C03580=1008.625,303.461,-161.555,-20.052,46.107,35.019
C03581=1008.519,303.701,-161.743,-19.485,46.587,36.235
C03582=1008.413,303.937,-161.933,-18.890,47.066,37.479
C03583=1008.305,304.173,-162.124,-18.265,47.545,38.750
C03584=1008.220,304.356,-162.274,-17.761,47.914,39.754
C03585=1008.136,304.538,-162.423,-17.237,48.283,40.777
C03586=1008.050,304.719,-162.574,-16.695,48.650,41.816
C03587=1007.964,304.899,-162.726,-16.132,49.015,42.875
C03588=1007.851,305.131,-162.923,-15.372,49.485,44.275
C03589=1007.738,305.362,-163.122,-14.578,49.950,45.708
C03590=1007.623,305.592,-163.322,-13.751,50.408,47.169
C03591=1007.508,305.821,-163.524,-12.888,50.859,48.662
C03592=1007.418,305.995,-163.679,-12.202,51.199,49.829
C03593=1007.328,306.169,-163.835,-11.496,51.534,51.012
C03594=1007.237,306.341,-163.992,-10.767,51.863,52.216
C03595=1007.147,306.513,-164.150,-10.017,52.187,53.438
C03596=1007.025,306.737,-164.358,-9.002,52.599,55.068
C03597=1006.905,306.961,-164.566,-7.948,53.000,56.733
C03598=1006.782,307.182,-164.777,-6.854,53.388,58.434
C03599=1006.659,307.402,-164.988,-5.724,53.761,60.165
C03600=1006.565,307.568,-165.150,-4.837,54.035,61.506
C03601=1006.470,307.733,-165.312,-3.930,54.299,62.863
C03602=1006.375,307.898,-165.475,-2.999,54.554,64.242
C03603=1006.278,308.061,-165.638,-2.047,54.798,65.640
C03604=1006.150,308.276,-165.856,-0.758,55.103,67.512
C03605=1006.021,308.489,-166.075,0.564,55.388,69.411
C03606=1005.891,308.702,-166.295,1.921,55.651,71.337
C03607=1005.760,308.912,-166.516,3.305,55.891,73.285
C03608=1005.653,309.083,-166.696,4.453,56.070,74.887
C03609=1005.546,309.251,-166.878,5.620,56.233,76.503
C03610=1005.908,309.402,-167.279,6.450,56.338,77.647
C03611=1006.056,309.174,-167.035,4.862,56.129,75.455
C03612=1006.201,308.944,-166.790,3.305,55.891,73.285
C03613=1006.331,308.733,-166.569,1.921,55.651,71.337
C03614=1006.462,308.522,-166.350,0.564,55.388,69.411
C03615=1006.591,308.308,-166.131,-0.758,55.103,67.512
C03616=1006.719,308.092,-165.913,-2.047,54.798,65.640
C03617=1006.815,307.929,-165.750,-2.999,54.554,64.242
C03618=1006.910,307.765,-165.587,-3.930,54.299,62.863
C03619=1007.005,307.600,-165.425,-4.837,54.035,61.506
C03620=1007.099,307.434,-165.263,-5.724,53.761,60.165
C03621=1007.223,307.214,-165.051,-6.854,53.388,58.434
C03622=1007.345,306.992,-164.841,-7.948,53.000,56.733
C03623=1007.467,306.769,-164.632,-9.002,52.599,55.068
C03624=1007.587,306.545,-164.424,-10.017,52.187,53.438
C03625=1007.677,306.373,-164.267,-10.767,51.863,52.216
C03626=1007.768,306.200,-164.110,-11.496,51.534,51.012
C03627=1007.858,306.027,-163.954,-12.202,51.199,49.829
C03628=1007.948,305.853,-163.798,-12.888,50.859,48.662
C03629=1008.064,305.623,-163.596,-13.751,50.408,47.169
C03630=1008.178,305.394,-163.396,-14.578,49.950,45.708
C03631=1008.291,305.163,-163.197,-15.372,49.485,44.275
C03632=1008.404,304.930,-163.000,-16.132,49.015,42.875
C03633=1008.490,304.750,-162.849,-16.695,48.650,41.816
C03634=1008.576,304.569,-162.698,-17.237,48.283,40.777
C03635=1008.661,304.388,-162.548,-17.761,47.914,39.754
C03636=1008.745,304.206,-162.398,-18.265,47.545,38.750
C03637=1008.853,303.969,-162.207,-18.890,47.066,37.479
C03638=1008.959,303.732,-162.018,-19.485,46.587,36.235
C03639=1009.065,303.494,-161.829,-20.052,46.107,35.019
C03640=1009.170,303.254,-161.642,-20.592,45.628,33.828
C03641=1009.251,303.066,-161.497,-20.996,45.254,32.916
C03642=1009.330,302.878,-161.352,-21.384,44.880,32.017
C03643=1009.410,302.689,-161.209,-21.757,44.508,31.133
C03644=1009.490,302.499,-161.066,-22.115,44.137,30.264
C03645=1009.590,302.256,-160.886,-22.552,43.665,29.173
C03646=1009.689,302.013,-160.706,-22.967,43.196,28.105
C03647=1009.787,301.768,-160.527,-23.359,42.732,27.060
C03648=1009.884,301.522,-160.351,-23.731,42.271,26.037
C03649=1009.959,301.327,-160.212,-24.010,41.911,25.245
C03650=1010.035,301.132,-160.075,-24.278,41.553,24.463
C03651=1010.110,300.936,-159.937,-24.533,41.199,23.695
C03652=1010.183,300.739,-159.802,-24.778,40.847,22.938
C03653=1010.276,300.491,-159.630,-25.071,40.409,21.999
C03654=1010.367,300.241,-159.461,-25.349,39.974,21.077
C03655=1010.458,299.990,-159.293,-25.610,39.546,20.172
///RCONF 0,0,0,0,1,0,0,0,0,0,0,0,0,0,0,0,0,0,0,0,0,0,0,0
C03656=1010.548,299.739,-159.127,-25.857,39.121,19.283
C03657=1010.618,299.539,-158.994,-26.044,38.788,18.586
C03658=1010.688,299.336,-158.863,-26.221,38.458,17.898
C03659=1010.757,299.135,-158.733,-26.391,38.132,17.220
C03660=1010.826,298.932,-158.604,-26.551,37.810,16.553
C03661=1010.911,298.678,-158.442,-26.741,37.414,15.733
C03662=1010.996,298.423,-158.283,-26.918,37.024,14.926
C03663=1011.079,298.168,-158.125,-27.085,36.641,14.134
C03664=1011.161,297.911,-157.968,-27.241,36.263,13.354
C03665=1011.228,297.705,-157.842,-27.359,35.965,12.738
C03666=1011.293,297.498,-157.718,-27.470,35.670,12.129
C03667=1011.357,297.290,-157.593,-27.576,35.380,11.529
C03668=1011.421,297.082,-157.470,-27.675,35.094,10.935
C03669=1011.499,296.824,-157.319,-27.790,34.746,10.213
C03670=1011.577,296.565,-157.169,-27.897,34.404,9.500
C03671=1011.653,296.305,-157.020,-27.996,34.069,8.801
C03672=1011.729,296.045,-156.872,-28.087,33.739,8.111
C03673=1011.789,295.834,-156.753,-28.156,33.478,7.560
C03674=1011.850,295.621,-156.636,-28.220,33.220,7.016
C03675=1011.910,295.408,-156.517,-28.280,32.966,6.479
C03676=1011.969,295.196,-156.400,-28.335,32.716,5.947
C03677=1012.041,294.934,-156.258,-28.398,32.417,5.306
C03678=1012.112,294.670,-156.117,-28.455,32.122,4.672
C03679=1012.182,294.408,-155.978,-28.506,31.835,4.050
C03680=1012.252,294.143,-155.838,-28.552,31.552,3.436
C03681=1012.308,293.928,-155.725,-28.586,31.327,2.940
C03682=1012.364,293.711,-155.613,-28.617,31.104,2.450
C03683=1012.419,293.493,-155.501,-28.645,30.886,1.967
C03684=1012.473,293.276,-155.391,-28.669,30.673,1.490
C03685=1012.539,293.010,-155.257,-28.695,30.417,0.916
C03686=1012.603,292.745,-155.124,-28.717,30.168,0.353
C03687=1012.668,292.479,-154.993,-28.736,29.926,-0.203
C03688=1012.731,292.212,-154.862,-28.751,29.686,-0.753
C03689=1012.783,291.992,-154.755,-28.760,29.494,-1.200
C03690=1012.834,291.771,-154.649,-28.768,29.306,-1.642
C03691=1012.885,291.550,-154.543,-28.773,29.120,-2.080
C03692=1012.935,291.329,-154.438,-28.777,28.937,-2.514
C03693=1012.996,291.061,-154.312,-28.778,28.722,-3.030
C03694=1013.054,290.793,-154.187,-28.777,28.512,-3.541
C03695=1013.113,290.524,-154.064,-28.773,28.305,-4.046
C03696=1013.171,290.255,-153.941,-28.767,28.103,-4.544
C03697=1013.219,290.031,-153.840,-28.760,27.939,-4.952
C03698=1013.265,289.806,-153.739,-28.752,27.779,-5.357
C03699=1013.312,289.582,-153.639,-28.742,27.622,-5.757
C03700=1013.358,289.357,-153.540,-28.730,27.467,-6.153
C03701=1013.413,289.087,-153.422,-28.715,27.285,-6.624
C03702=1013.467,288.817,-153.304,-28.698,27.109,-7.088
C03703=1013.520,288.545,-153.189,-28.679,26.937,-7.545
C03704=1013.573,288.274,-153.072,-28.659,26.767,-7.999
C03705=1013.617,288.047,-152.977,-28.641,26.630,-8.372
C03706=1013.660,287.819,-152.882,-28.622,26.495,-8.743
C03707=1013.701,287.592,-152.787,-28.602,26.363,-9.109
C03708=1013.744,287.364,-152.694,-28.581,26.233,-9.471
C03709=1013.794,287.092,-152.582,-28.555,26.082,-9.899
C03710=1013.842,286.820,-152.472,-28.527,25.935,-10.321
C03711=1013.890,286.547,-152.363,-28.499,25.792,-10.737
C03712=1013.938,286.275,-152.254,-28.470,25.652,-11.148
C03713=1013.978,286.044,-152.164,-28.444,25.537,-11.492
C03714=1014.017,285.814,-152.074,-28.418,25.425,-11.832
C03715=1014.056,285.584,-151.985,-28.391,25.314,-12.171
C03716=1014.094,285.354,-151.895,-28.364,25.204,-12.507
C03717=1014.139,285.080,-151.791,-28.330,25.079,-12.901
C03718=1014.183,284.807,-151.688,-28.296,24.956,-13.292
C03719=1014.227,284.533,-151.585,-28.261,24.835,-13.680
C03720=1014.270,284.258,-151.484,-28.226,24.716,-14.065
C03721=1014.306,284.026,-151.398,-28.195,24.619,-14.388
C03722=1014.341,283.794,-151.313,-28.164,24.524,-14.708
C03723=1014.377,283.561,-151.229,-28.132,24.429,-15.026
C03724=1014.411,283.328,-151.145,-28.100,24.338,-15.343
C03725=1014.451,283.053,-151.048,-28.062,24.232,-15.713
C03726=1014.490,282.778,-150.950,-28.023,24.128,-16.079
C03727=1014.530,282.504,-150.854,-27.984,24.027,-16.441
C03728=1014.568,282.228,-150.759,-27.945,23.929,-16.801
C03729=1014.600,281.993,-150.677,-27.911,23.848,-17.104
C03730=1014.633,281.758,-150.597,-27.877,23.768,-17.406
C03731=1014.663,281.524,-150.518,-27.842,23.690,-17.706
C03732=1014.695,281.288,-150.439,-27.807,23.613,-18.004
C03733=1014.731,281.013,-150.347,-27.766,23.526,-18.349
C03734=1014.766,280.737,-150.256,-27.725,23.440,-18.691
C03735=1014.800,280.461,-150.166,-27.684,23.357,-19.031
C03736=1014.835,280.185,-150.076,-27.642,23.276,-19.367
C03737=1014.863,279.948,-150.000,-27.606,23.208,-19.653
C03738=1014.892,279.711,-149.925,-27.570,23.143,-19.936
C03739=1014.920,279.474,-149.851,-27.534,23.078,-20.218
C03740=1014.948,279.238,-149.777,-27.498,23.014,-20.499
C03741=1014.980,278.961,-149.691,-27.456,22.942,-20.824
C03742=1015.011,278.685,-149.606,-27.413,22.872,-21.148
C03743=1015.042,278.408,-149.522,-27.370,22.804,-21.469
C03744=1015.072,278.131,-149.437,-27.327,22.737,-21.789
C03745=1015.097,277.892,-149.366,-27.290,22.681,-22.062
C03746=1015.122,277.654,-149.296,-27.252,22.626,-22.334
C03747=1015.148,277.415,-149.226,-27.215,22.573,-22.606
C03748=1015.172,277.176,-149.155,-27.177,22.521,-22.877
C03749=1015.199,276.899,-149.076,-27.134,22.462,-23.186
C03750=1015.226,276.622,-148.996,-27.090,22.404,-23.496
C03751=1015.253,276.345,-148.917,-27.046,22.349,-23.804
C03752=1015.279,276.068,-148.840,-27.003,22.295,-24.109
C03753=1015.301,275.828,-148.773,-26.965,22.250,-24.373
C03754=1015.323,275.588,-148.708,-26.927,22.204,-24.635
C03755=1015.344,275.347,-148.641,-26.889,22.162,-24.896
C03756=1015.366,275.107,-148.577,-26.851,22.119,-25.156
C03757=1015.390,274.829,-148.502,-26.807,22.073,-25.453
C03758=1015.412,274.552,-148.428,-26.763,22.027,-25.750
C03759=1015.435,274.275,-148.355,-26.720,21.983,-26.043
C03760=1015.458,273.996,-148.282,-26.676,21.940,-26.336
C03761=1015.477,273.755,-148.221,-26.638,21.904,-26.589
C03762=1015.496,273.513,-148.158,-26.600,21.869,-26.841
C03763=1015.513,273.271,-148.097,-26.562,21.835,-27.092
C03764=1015.532,273.030,-148.036,-26.525,21.803,-27.342
C03765=1015.551,272.752,-147.968,-26.481,21.766,-27.626
C03766=1015.571,272.474,-147.900,-26.438,21.731,-27.910
C03767=1015.591,272.196,-147.832,-26.395,21.697,-28.194
C03768=1015.609,271.918,-147.764,-26.351,21.664,-28.476
C03769=1015.625,271.674,-147.706,-26.314,21.637,-28.720
C03770=1015.640,271.432,-147.649,-26.276,21.610,-28.964
C03771=1015.656,271.188,-147.593,-26.238,21.585,-29.208
C03772=1015.670,270.945,-147.536,-26.201,21.560,-29.450
C03773=1015.685,270.668,-147.472,-26.158,21.533,-29.728
C03774=1015.703,270.389,-147.409,-26.115,21.507,-30.003
C03775=1015.718,270.111,-147.348,-26.072,21.483,-30.277
C03776=1015.732,269.832,-147.286,-26.030,21.459,-30.551
C03777=1015.746,269.588,-147.232,-25.992,21.438,-30.791
C03778=1015.757,269.344,-147.180,-25.955,21.420,-31.029
C03779=1015.769,269.100,-147.127,-25.918,21.402,-31.266
C03780=1015.781,268.856,-147.075,-25.881,21.386,-31.502
C03781=1015.794,268.577,-147.017,-25.839,21.367,-31.772
C03782=1015.806,268.299,-146.958,-25.797,21.350,-32.039
C03783=1015.818,268.021,-146.901,-25.755,21.334,-32.305
C03784=1015.829,267.742,-146.845,-25.714,21.319,-32.571
C03785=1015.839,267.497,-146.796,-25.677,21.306,-32.805
C03786=1015.848,267.251,-146.747,-25.641,21.295,-33.037
C03787=1015.857,267.006,-146.699,-25.604,21.284,-33.268
C03788=1015.866,266.760,-146.652,-25.568,21.275,-33.499
C03789=1015.875,266.482,-146.599,-25.527,21.264,-33.760
C03790=1015.883,266.203,-146.545,-25.487,21.254,-34.021
C03791=1015.891,265.925,-146.493,-25.446,21.246,-34.279
C03792=1015.899,265.646,-146.442,-25.406,21.239,-34.538
C03793=1015.905,265.399,-146.398,-25.370,21.233,-34.766
C03794=1015.912,265.154,-146.353,-25.335,21.229,-34.991
C03795=1015.918,264.908,-146.310,-25.300,21.225,-35.219
C03796=1015.924,264.661,-146.267,-25.265,21.221,-35.444
C03797=1015.929,264.383,-146.219,-25.226,21.219,-35.699
C03798=1015.934,264.103,-146.170,-25.186,21.217,-35.952
C03799=1015.939,263.824,-146.124,-25.147,21.216,-36.205
C03800=1015.943,263.545,-146.078,-25.108,21.215,-36.458
C03801=1015.947,263.298,-146.037,-25.074,21.216,-36.681
C03802=1015.950,263.051,-145.997,-25.040,21.217,-36.903
C03803=1015.953,262.804,-145.958,-25.006,21.220,-37.124
C03804=1015.955,262.558,-145.919,-24.973,21.223,-37.345
C03805=1015.957,262.278,-145.876,-24.935,21.227,-37.593
C03806=1015.959,261.999,-145.833,-24.897,21.233,-37.842
C03807=1015.961,261.719,-145.791,-24.860,21.238,-38.090
C03808=1015.961,261.440,-145.750,-24.823,21.245,-38.337
C03809=1015.962,261.192,-145.714,-24.790,21.251,-38.554
C03810=1015.962,260.945,-145.679,-24.758,21.259,-38.770
C03811=1015.962,260.698,-145.644,-24.725,21.267,-38.988
C03812=1015.961,260.451,-145.609,-24.693,21.275,-39.204
C03813=1015.960,260.171,-145.571,-24.658,21.287,-39.446
C03814=1015.958,259.891,-145.533,-24.622,21.298,-39.688
C03815=1015.957,259.612,-145.496,-24.587,21.310,-39.930
C03816=1015.954,259.332,-145.460,-24.551,21.322,-40.171
C03817=1015.938,258.096,-145.307,-24.430,21.375,-41.012
C03818=1015.934,257.852,-145.277,-24.430,21.375,-41.014
C03819=1015.931,257.609,-145.248,-24.429,21.375,-41.018
C03820=1015.928,257.366,-145.220,-24.429,21.376,-41.019
C03821=1015.925,257.122,-145.191,-24.429,21.376,-41.021
C03822=1015.922,256.879,-145.162,-24.428,21.375,-41.025
C03823=1015.919,256.635,-145.132,-24.428,21.376,-41.027
C03824=1015.915,256.392,-145.104,-24.428,21.377,-41.029
C03825=1015.912,256.144,-145.074,-24.427,21.376,-41.032
C03826=1015.908,255.895,-145.044,-24.427,21.376,-41.034
C03827=1015.905,255.648,-145.014,-24.426,21.376,-41.037
C03828=1015.901,255.399,-144.985,-24.426,21.377,-41.040
C03829=1015.899,255.151,-144.955,-24.426,21.377,-41.042
C03830=1015.895,254.903,-144.926,-24.425,21.377,-41.045
C03831=1015.892,254.654,-144.897,-24.425,21.377,-41.047
C03832=1015.889,254.406,-144.866,-24.425,21.377,-41.049
C03833=1015.885,254.158,-144.837,-24.424,21.378,-41.052
C03834=1015.882,253.909,-144.808,-24.424,21.378,-41.054
C03835=1015.879,253.661,-144.779,-24.424,21.378,-41.058
C03836=1015.876,253.414,-144.749,-24.423,21.378,-41.060
C03837=1015.872,253.165,-144.720,-24.423,21.378,-41.061
C03838=1015.870,252.917,-144.690,-24.423,21.378,-41.065
C03839=1015.866,252.668,-144.660,-24.422,21.379,-41.067
C03840=1015.863,252.420,-144.631,-24.422,21.379,-41.069
C03841=1015.860,252.172,-144.602,-24.421,21.378,-41.072
C03842=1015.857,251.923,-144.572,-24.421,21.379,-41.074
C03843=1015.854,251.675,-144.544,-24.421,21.380,-41.076
C03844=1015.850,251.427,-144.513,-24.421,21.380,-41.078
C03845=1015.847,251.184,-144.485,-24.420,21.380,-41.082
C03846=1015.844,250.940,-144.456,-24.420,21.380,-41.084
C03847=1015.841,250.697,-144.428,-24.420,21.380,-41.085
C03848=1015.838,250.454,-144.399,-24.419,21.380,-41.089
C03849=1015.835,250.211,-144.370,-24.419,21.380,-41.091
C03850=1015.831,249.968,-144.341,-24.419,21.381,-41.093
C03851=1015.829,249.724,-144.313,-24.418,21.381,-41.095
C03852=1015.826,249.480,-144.284,-24.418,21.381,-41.098
C03853=1015.823,249.232,-144.255,-24.418,21.381,-41.100
C03854=1015.819,248.984,-144.226,-24.417,21.381,-41.102
C03855=1015.816,248.735,-144.197,-24.417,21.381,-41.104
C03856=1015.813,248.488,-144.168,-24.417,21.381,-41.107
C03857=1015.810,248.240,-144.138,-24.416,21.381,-41.109
C03858=1015.807,247.992,-144.109,-24.416,21.382,-41.111
C03859=1015.804,247.743,-144.079,-24.416,21.382,-41.113
C03860=1015.800,247.495,-144.051,-24.415,21.382,-41.117
C03861=1015.798,247.247,-144.021,-24.415,21.382,-41.118
C03862=1015.795,246.999,-143.992,-24.415,21.382,-41.120
C03863=1015.792,246.750,-143.964,-24.414,21.383,-41.122
C03864=1015.789,246.501,-143.935,-24.414,21.382,-41.126
C03865=1015.786,246.253,-143.905,-24.414,21.382,-41.127
C03866=1015.783,246.005,-143.876,-24.413,21.383,-41.129
C03867=1015.780,245.757,-143.847,-24.413,21.384,-41.132
C03868=1015.777,245.509,-143.818,-24.413,21.384,-41.134
C03869=1015.773,245.260,-143.789,-24.412,21.384,-41.137
C03870=1015.771,245.012,-143.760,-24.412,21.384,-41.139
C03871=1015.767,244.764,-143.731,-24.412,21.384,-41.141
C03872=1015.765,244.515,-143.702,-24.412,21.384,-41.143
C03873=1015.762,244.279,-143.674,-24.411,21.384,-41.144
C03874=1015.759,244.041,-143.647,-24.411,21.384,-41.148
C03875=1015.756,243.804,-143.620,-24.411,21.384,-41.150
C03876=1015.754,243.567,-143.591,-24.410,21.384,-41.151
C03877=1015.751,243.330,-143.564,-24.410,21.385,-41.153
C03878=1015.748,243.093,-143.536,-24.410,21.385,-41.155
C03879=1015.745,242.857,-143.509,-24.410,21.385,-41.157
C03880=1015.742,242.619,-143.481,-24.409,21.385,-41.159
C03881=1015.739,242.371,-143.452,-24.409,21.386,-41.161
C03882=1015.736,242.123,-143.423,-24.408,21.385,-41.164
C03883=1015.734,241.874,-143.394,-24.408,21.385,-41.166
C03884=1015.731,241.626,-143.365,-24.408,21.386,-41.168
C03885=1015.728,241.378,-143.336,-24.408,21.386,-41.170
C03886=1015.725,241.129,-143.308,-24.407,21.386,-41.172
C03887=1015.723,240.881,-143.279,-24.407,21.386,-41.174
C03888=1015.719,240.633,-143.250,-24.407,21.386,-41.176
C03889=1015.717,240.385,-143.222,-24.406,21.386,-41.179
C03890=1015.714,240.136,-143.192,-24.406,21.386,-41.181
C03891=1015.711,239.888,-143.164,-24.406,21.386,-41.183
C03892=1015.709,239.639,-143.135,-24.406,21.387,-41.184
C03893=1015.706,239.379,-143.105,-24.405,21.387,-41.186
C03894=1015.702,239.118,-143.075,-24.405,21.387,-41.188
C03895=1015.699,238.858,-143.044,-24.405,21.387,-41.190
C03896=1015.696,238.597,-143.014,-24.405,21.388,-41.192
C03897=1015.694,238.348,-142.986,-24.404,21.387,-41.195
C03898=1015.691,238.100,-142.957,-24.404,21.387,-41.197
C03899=1015.688,237.852,-142.929,-24.403,21.388,-41.199
C03900=1015.686,237.604,-142.900,-24.403,21.388,-41.201
C03901=1015.683,237.360,-142.872,-24.403,21.388,-41.203
C03902=1015.680,237.117,-142.843,-24.403,21.388,-41.205
C03903=1015.677,236.874,-142.816,-24.402,21.388,-41.207
C03904=1015.675,236.631,-142.787,-24.402,21.389,-41.209
C03905=1015.672,236.388,-142.759,-24.402,21.389,-41.210
C03906=1015.670,236.145,-142.731,-24.402,21.389,-41.212
C03907=1015.667,235.902,-142.704,-24.401,21.389,-41.214
C03908=1015.664,235.659,-142.676,-24.401,21.390,-41.216
C03909=1015.662,235.410,-142.647,-24.401,21.389,-41.218
C03910=1015.658,235.162,-142.618,-24.401,21.389,-41.219
C03911=1015.656,234.914,-142.589,-24.400,21.389,-41.221
C03912=1015.653,234.665,-142.561,-24.400,21.390,-41.223
C03913=1015.651,234.418,-142.533,-24.400,21.390,-41.225
C03914=1015.648,234.169,-142.504,-24.400,21.390,-41.227
C03915=1015.645,233.921,-142.475,-24.399,21.390,-41.229
C03916=1015.643,233.672,-142.447,-24.399,21.390,-41.231
C03917=1015.640,233.423,-142.419,-24.399,21.391,-41.233
C03918=1015.638,233.176,-142.390,-24.399,21.391,-41.234
C03919=1015.635,232.927,-142.362,-24.398,21.391,-41.236
C03920=1015.632,232.679,-142.334,-24.398,21.390,-41.238
C03921=1015.630,232.430,-142.304,-24.398,21.391,-41.240
C03922=1015.627,232.182,-142.277,-24.397,21.391,-41.242
C03923=1015.625,231.933,-142.248,-24.397,21.391,-41.243
C03924=1015.622,231.685,-142.220,-24.397,21.391,-41.245
C03925=1015.619,231.437,-142.191,-24.397,21.392,-41.247
C03926=1015.617,231.189,-142.163,-24.396,21.392,-41.249
C03927=1015.614,230.940,-142.135,-24.396,21.392,-41.251
C03928=1015.612,230.691,-142.106,-24.396,21.391,-41.252
C03929=1015.609,230.449,-142.078,-24.396,21.392,-41.254
C03930=1015.607,230.206,-142.050,-24.395,21.392,-41.256
C03931=1015.605,229.963,-142.023,-24.395,21.392,-41.258
C03932=1015.602,229.720,-141.995,-24.395,21.392,-41.260
C03933=1015.600,229.476,-141.967,-24.395,21.392,-41.262
C03934=1015.597,229.234,-141.940,-24.394,21.392,-41.263
C03935=1015.594,228.991,-141.912,-24.394,21.392,-41.265
C03936=1015.593,228.748,-141.885,-24.394,21.393,-41.266
C03937=1015.589,228.500,-141.856,-24.394,21.393,-41.267
C03938=1015.588,228.252,-141.827,-24.394,21.393,-41.269
C03939=1015.585,228.003,-141.799,-24.393,21.394,-41.271
C03940=1015.582,227.755,-141.771,-24.393,21.393,-41.273
C03941=1015.580,227.506,-141.743,-24.393,21.393,-41.275
C03942=1015.577,227.258,-141.715,-24.393,21.393,-41.276
C03943=1015.576,227.010,-141.687,-24.392,21.394,-41.278
C03944=1015.573,226.761,-141.659,-24.392,21.394,-41.280
C03945=1015.570,226.512,-141.631,-24.392,21.393,-41.282
C03946=1015.568,226.264,-141.602,-24.391,21.393,-41.284
C03947=1015.565,226.016,-141.574,-24.391,21.394,-41.285
C03948=1015.563,225.767,-141.546,-24.391,21.395,-41.286
C03949=1015.560,225.519,-141.518,-24.391,21.395,-41.288
C03950=1015.559,225.271,-141.490,-24.391,21.394,-41.289
C03951=1015.556,225.022,-141.461,-24.390,21.394,-41.291
C03952=1015.554,224.774,-141.434,-24.390,21.395,-41.293
C03953=1015.551,224.525,-141.405,-24.390,21.395,-41.295
C03954=1015.548,224.277,-141.377,-24.390,21.395,-41.297
C03955=1015.547,224.028,-141.349,-24.389,21.394,-41.298
C03956=1015.544,223.780,-141.321,-24.389,21.395,-41.300
C03957=1015.541,223.537,-141.293,-24.389,21.395,-41.300
C03958=1015.540,223.294,-141.266,-24.389,21.396,-41.302
C03959=1015.537,223.052,-141.239,-24.389,21.396,-41.304
C03960=1015.534,222.809,-141.211,-24.388,21.395,-41.306
C03961=1015.533,222.566,-141.183,-24.388,21.395,-41.308
C03962=1015.531,222.323,-141.156,-24.388,21.396,-41.309
C03963=1015.528,222.081,-141.129,-24.388,21.397,-41.310
C03964=1015.526,221.838,-141.102,-24.388,21.396,-41.311
C03965=1015.524,221.589,-141.074,-24.387,21.396,-41.313
C03966=1015.522,221.341,-141.046,-24.387,21.396,-41.315
C03967=1015.519,221.092,-141.017,-24.387,21.397,-41.317
C03968=1015.517,220.844,-140.990,-24.386,21.396,-41.318
C03969=1015.514,220.596,-140.962,-24.386,21.396,-41.320
C03970=1015.512,220.347,-140.933,-24.386,21.397,-41.321
C03971=1015.510,220.098,-140.906,-24.386,21.397,-41.323
C03972=1015.508,219.850,-140.878,-24.386,21.397,-41.324
C03973=1015.506,219.602,-140.850,-24.385,21.397,-41.326
C03974=1015.503,219.353,-140.822,-24.385,21.397,-41.328
C03975=1015.501,219.105,-140.794,-24.385,21.397,-41.330
C03976=1015.499,218.857,-140.767,-24.385,21.397,-41.330
C03977=1015.497,218.608,-140.738,-24.385,21.397,-41.332
C03978=1015.495,218.360,-140.710,-24.384,21.398,-41.333
C03979=1015.493,218.111,-140.683,-24.384,21.398,-41.335
C03980=1015.490,217.863,-140.655,-24.384,21.397,-41.337
C03981=1015.488,217.615,-140.627,-24.384,21.397,-41.339
C03982=1015.487,217.366,-140.599,-24.384,21.398,-41.339
C03983=1015.484,217.117,-140.571,-24.383,21.399,-41.341
C03984=1015.482,216.869,-140.543,-24.383,21.398,-41.342
C03985=1015.480,216.627,-140.516,-24.383,21.398,-41.344
C03986=1015.478,216.383,-140.489,-24.383,21.398,-41.346
C03987=1015.475,216.141,-140.462,-24.383,21.398,-41.346
C03988=1015.474,215.898,-140.434,-24.382,21.399,-41.348
C03989=1015.471,215.655,-140.407,-24.382,21.399,-41.350
C03990=1015.469,215.412,-140.381,-24.382,21.399,-41.352
C03991=1015.467,215.170,-140.353,-24.382,21.398,-41.353
C03992=1015.465,214.927,-140.326,-24.382,21.399,-41.354
C03993=1015.463,214.678,-140.299,-24.381,21.400,-41.356
C03994=1015.461,214.431,-140.271,-24.381,21.399,-41.357
C03995=1015.459,214.182,-140.243,-24.381,21.399,-41.359
C03996=1015.457,213.933,-140.215,-24.381,21.400,-41.359
C03997=1015.455,213.685,-140.187,-24.381,21.400,-41.361
C03998=1015.453,213.436,-140.160,-24.380,21.400,-41.363
C03999=1015.450,213.189,-140.132,-24.380,21.400,-41.365
C04000=1015.449,212.940,-140.105,-24.380,21.400,-41.366
C04001=1015.446,212.691,-140.077,-24.380,21.400,-41.366
C04002=1015.445,212.442,-140.049,-24.380,21.400,-41.368
C04003=1015.443,212.194,-140.021,-24.379,21.400,-41.370
C04004=1015.440,211.946,-139.994,-24.379,21.400,-41.372
C04005=1015.439,211.698,-139.966,-24.379,21.401,-41.372
C04006=1015.436,211.449,-139.939,-24.379,21.401,-41.374
C04007=1015.435,211.200,-139.910,-24.378,21.400,-41.375
C04008=1015.433,210.952,-139.883,-24.378,21.400,-41.377
C04009=1015.431,210.703,-139.856,-24.378,21.401,-41.378
C04010=1015.429,210.455,-139.828,-24.378,21.401,-41.379
C04011=1015.427,210.207,-139.801,-24.378,21.401,-41.381
C04012=1015.425,209.958,-139.773,-24.377,21.401,-41.383
C04013=1015.423,209.715,-139.746,-24.377,21.401,-41.383
C04014=1015.421,209.473,-139.719,-24.377,21.401,-41.385
C04015=1015.419,209.230,-139.693,-24.377,21.402,-41.387
C04016=1015.418,208.987,-139.665,-24.377,21.401,-41.388
C04017=1015.416,208.744,-139.639,-24.377,21.402,-41.389
C04018=1015.414,208.503,-139.612,-24.376,21.402,-41.391
C04019=1015.412,208.260,-139.585,-24.376,21.401,-41.392
C04020=1015.409,208.017,-139.558,-24.376,21.402,-41.392
C04021=1015.408,207.768,-139.531,-24.376,21.402,-41.394
C04022=1015.406,207.520,-139.503,-24.376,21.402,-41.396
C04023=1015.404,207.271,-139.476,-24.375,21.402,-41.398
C04024=1015.402,207.023,-139.449,-24.375,21.402,-41.398
C04025=1015.400,206.775,-139.421,-24.375,21.402,-41.399
C04026=1015.399,206.526,-139.393,-24.375,21.402,-41.401
C04027=1015.397,206.278,-139.366,-24.375,21.402,-41.401
C04028=1015.395,206.029,-139.339,-24.375,21.403,-41.403
C04029=1015.393,205.781,-139.311,-24.374,21.403,-41.405
C04030=1015.392,205.532,-139.283,-24.374,21.402,-41.407
C04031=1015.390,205.284,-139.256,-24.374,21.403,-41.407
C04032=1015.388,205.035,-139.229,-24.374,21.403,-41.409
C04033=1015.386,204.787,-139.201,-24.373,21.403,-41.410
C04034=1015.384,204.538,-139.174,-24.374,21.404,-41.411
C04035=1015.383,204.290,-139.147,-24.373,21.403,-41.412
C04036=1015.381,204.041,-139.120,-24.373,21.403,-41.414
C04037=1015.379,203.792,-139.093,-24.373,21.404,-41.415
C04038=1015.377,203.544,-139.064,-24.373,21.403,-41.416
C04039=1015.372,202.328,-138.930,-24.425,21.378,-41.051
C04040=1015.371,201.941,-138.886,-24.424,21.378,-41.052
C04041=1015.372,201.592,-138.848,-24.424,21.378,-41.054
C04042=1015.373,201.240,-138.809,-24.424,21.378,-41.058
C04043=1015.374,200.833,-138.765,-24.423,21.379,-41.060
C04044=1015.374,200.606,-138.740,-24.423,21.378,-41.061
C04045=1015.374,200.377,-138.715,-24.423,21.378,-41.063
C04046=1015.374,200.154,-138.690,-24.423,21.378,-41.065
C04047=1015.375,199.942,-138.667,-24.423,21.378,-41.065
C04048=1015.375,199.541,-138.623,-24.422,21.379,-41.069
C04049=1015.377,199.151,-138.582,-24.422,21.379,-41.071
C04050=1015.377,198.753,-138.538,-24.421,21.379,-41.074
C04051=1015.378,198.352,-138.493,-24.421,21.379,-41.076
C04052=1015.379,197.951,-138.450,-24.421,21.380,-41.078
C04053=1015.380,197.550,-138.407,-24.420,21.380,-41.082
C04054=1015.381,197.149,-138.362,-24.420,21.380,-41.084
C04055=1015.382,196.748,-138.319,-24.419,21.380,-41.087
C04056=1015.383,196.346,-138.276,-24.419,21.380,-41.089
C04057=1015.383,195.946,-138.232,-24.419,21.381,-41.091
C04058=1015.384,195.544,-138.188,-24.418,21.380,-41.094
C04059=1015.385,195.143,-138.144,-24.418,21.381,-41.097
C04060=1015.386,194.742,-138.101,-24.418,21.381,-41.100
C04061=1015.387,194.341,-138.058,-24.417,21.381,-41.102
C04062=1015.388,193.940,-138.013,-24.417,21.381,-41.105
C04063=1015.389,193.539,-137.970,-24.417,21.382,-41.108
C04064=1015.389,193.137,-137.926,-24.416,21.382,-41.109
C04065=1015.391,192.737,-137.884,-24.416,21.382,-41.113
C04066=1015.391,192.336,-137.840,-24.415,21.382,-41.115
C04067=1015.393,191.934,-137.796,-24.415,21.382,-41.118
C04068=1015.394,191.533,-137.753,-24.415,21.382,-41.120
C04069=1015.394,191.132,-137.710,-24.414,21.382,-41.124
C04070=1015.396,190.731,-137.667,-24.414,21.383,-41.126
C04071=1015.397,190.330,-137.623,-24.414,21.383,-41.128
C04072=1015.398,189.928,-137.579,-24.413,21.383,-41.131
C04073=1015.399,189.528,-137.537,-24.413,21.383,-41.133
C04074=1015.400,189.127,-137.493,-24.412,21.384,-41.137
C04075=1015.401,188.725,-137.450,-24.412,21.384,-41.139
C04076=1015.402,188.324,-137.407,-24.412,21.384,-41.141
C04077=1015.403,187.924,-137.364,-24.411,21.384,-41.144
C04078=1015.404,187.522,-137.320,-24.411,21.385,-41.146
C04079=1015.406,187.122,-137.277,-24.411,21.384,-41.150
C04080=1015.407,186.720,-137.233,-24.410,21.384,-41.151
C04081=1015.407,186.319,-137.190,-24.410,21.384,-41.155
C04082=1015.409,185.919,-137.147,-24.410,21.385,-41.157
C04083=1015.409,185.518,-137.104,-24.409,21.385,-41.159
C04084=1015.411,185.117,-137.061,-24.409,21.385,-41.162
C04085=1015.412,184.715,-137.018,-24.409,21.386,-41.165
C04086=1015.413,184.315,-136.975,-24.408,21.386,-41.168
C04087=1015.414,183.913,-136.932,-24.408,21.386,-41.170
C04088=1015.415,183.513,-136.889,-24.407,21.386,-41.172
C04089=1015.417,183.112,-136.846,-24.407,21.386,-41.176
C04090=1015.418,182.711,-136.804,-24.407,21.387,-41.177
C04091=1015.419,182.310,-136.761,-24.406,21.386,-41.181
C04092=1015.420,181.910,-136.718,-24.406,21.387,-41.183
C04093=1015.421,181.508,-136.674,-24.405,21.387,-41.186
C04094=1015.423,181.107,-136.632,-24.405,21.387,-41.188
C04095=1015.424,180.707,-136.589,-24.405,21.387,-41.190
C04096=1015.425,180.306,-136.546,-24.404,21.388,-41.194
C04097=1015.426,179.905,-136.503,-24.404,21.388,-41.196
C04098=1015.428,179.504,-136.461,-24.403,21.388,-41.199
C04099=1015.429,179.103,-136.418,-24.403,21.388,-41.201
C04100=1015.430,178.702,-136.374,-24.403,21.388,-41.205
C04101=1015.432,178.301,-136.332,-24.402,21.388,-41.207
C04102=1015.433,177.901,-136.289,-24.402,21.389,-41.209
C04103=1015.434,177.500,-136.246,-24.402,21.389,-41.212
C04104=1015.435,177.099,-136.205,-24.401,21.389,-41.214
C04105=1015.437,176.699,-136.162,-24.401,21.389,-41.218
C04106=1015.438,176.298,-136.119,-24.401,21.389,-41.219
C04107=1015.440,175.897,-136.077,-24.400,21.390,-41.223
C04108=1015.441,175.497,-136.034,-24.400,21.390,-41.225
C04109=1015.443,175.095,-135.991,-24.400,21.390,-41.227
C04110=1015.443,174.695,-135.949,-24.399,21.390,-41.231
C04111=1015.445,174.295,-135.906,-24.399,21.391,-41.233
C04112=1015.446,173.894,-135.864,-24.398,21.390,-41.236
C04113=1015.448,173.493,-135.821,-24.398,21.390,-41.238
C04114=1015.449,173.092,-135.779,-24.397,21.391,-41.242
C04115=1015.450,172.692,-135.736,-24.397,21.391,-41.243
C04116=1015.451,172.291,-135.694,-24.397,21.391,-41.247
C04117=1015.453,171.890,-135.651,-24.396,21.392,-41.249
C04118=1015.455,171.490,-135.609,-24.396,21.392,-41.251
C04119=1015.456,171.090,-135.567,-24.396,21.392,-41.254
C04120=1015.457,170.689,-135.524,-24.395,21.392,-41.256
C04121=1015.459,170.288,-135.482,-24.395,21.392,-41.260
C04122=1015.459,169.888,-135.439,-24.395,21.392,-41.262
C04123=1015.462,169.487,-135.398,-24.394,21.392,-41.265
C04124=1015.463,169.087,-135.355,-24.394,21.393,-41.267
C04125=1015.464,168.686,-135.313,-24.393,21.393,-41.271
C04126=1015.466,168.286,-135.270,-24.393,21.393,-41.273
C04127=1015.467,167.885,-135.229,-24.393,21.394,-41.275
C04128=1015.468,167.484,-135.186,-24.392,21.394,-41.278
C04129=1015.470,167.084,-135.144,-24.392,21.394,-41.280
C04130=1015.471,166.684,-135.102,-24.391,21.393,-41.284
C04131=1015.473,166.284,-135.060,-24.391,21.395,-41.286
C04132=1015.474,165.883,-135.018,-24.391,21.394,-41.289
C04133=1015.476,165.483,-134.975,-24.390,21.394,-41.291
C04134=1015.477,165.082,-134.934,-24.390,21.395,-41.295
C04135=1015.479,164.683,-134.891,-24.390,21.395,-41.297
C04136=1015.480,164.283,-134.850,-24.389,21.395,-41.300
C04137=1015.482,163.896,-134.810,-24.389,21.395,-41.302
C04138=1015.483,163.706,-134.789,-24.389,21.395,-41.304
C04139=1015.484,163.294,-134.746,-24.388,21.396,-41.306
C04140=1015.484,163.059,-134.721,-24.388,21.395,-41.308
C04141=1015.486,162.805,-134.695,-24.388,21.396,-41.309
C04142=1015.487,162.542,-134.667,-24.388,21.396,-41.311
C04143=1015.488,162.273,-134.639,-24.387,21.396,-41.313
C04144=1015.489,162.002,-134.610,-24.387,21.396,-41.315
C04145=1015.489,161.733,-134.582,-24.387,21.397,-41.317
C04146=1015.491,161.470,-134.555,-24.387,21.397,-41.319
C04147=1015.492,161.219,-134.528,-24.386,21.396,-41.320
C04148=1015.492,160.982,-134.504,-24.386,21.396,-41.322
C04149=1015.494,160.757,-134.480,-24.386,21.397,-41.324
C04150=1015.495,160.544,-134.458,-24.386,21.397,-41.325
C04151=1015.496,160.139,-134.416,-24.385,21.397,-41.328
C04152=1015.497,159.742,-134.374,-24.385,21.397,-41.330
C04153=1015.505,159.342,-134.336,-24.384,21.398,-41.333
C04154=1015.512,158.942,-134.298,-24.384,21.398,-41.335
C04155=1015.520,158.540,-134.260,-24.384,21.397,-41.339
C04156=1015.527,158.138,-134.221,-24.383,21.399,-41.341
C04157=1015.534,157.736,-134.182,-24.383,21.398,-41.344
C04158=1015.542,157.332,-134.144,-24.383,21.398,-41.346
C04159=1015.550,156.928,-134.106,-24.382,21.399,-41.350
C04160=1015.557,156.523,-134.067,-24.382,21.399,-41.352
C04161=1015.564,156.118,-134.029,-24.381,21.399,-41.355
C04162=1015.571,155.711,-133.990,-24.381,21.400,-41.358
C04163=1015.579,155.303,-133.951,-24.381,21.399,-41.361
C04164=1015.586,154.895,-133.912,-24.380,21.400,-41.363
C04165=1015.594,154.486,-133.873,-24.380,21.400,-41.366
C04166=1015.601,154.076,-133.834,-24.380,21.400,-41.368
C04167=1015.608,153.665,-133.795,-24.379,21.401,-41.372
C04168=1015.615,153.254,-133.756,-24.378,21.400,-41.375
C04169=1015.623,152.842,-133.717,-24.378,21.400,-41.377
C04170=1015.631,152.430,-133.677,-24.378,21.401,-41.381
C04171=1015.638,152.018,-133.637,-24.377,21.401,-41.383
C04172=1015.645,151.604,-133.599,-24.377,21.402,-41.387
C04173=1015.652,151.191,-133.559,-24.377,21.402,-41.389
C04174=1015.659,150.777,-133.520,-24.376,21.401,-41.392
C04175=1015.667,150.364,-133.480,-24.376,21.402,-41.394
C04176=1015.673,149.950,-133.441,-24.375,21.402,-41.398
C04177=1015.681,149.536,-133.402,-24.375,21.402,-41.401
C04178=1015.688,149.122,-133.363,-24.375,21.403,-41.403
C04179=1015.695,148.709,-133.323,-24.374,21.403,-41.407
C04180=1015.702,148.294,-133.284,-24.374,21.403,-41.409
C04181=1015.709,147.880,-133.245,-24.373,21.403,-41.412
C04182=1015.716,147.467,-133.205,-24.373,21.403,-41.416
C04183=1015.724,147.053,-133.165,-24.372,21.404,-41.418
C04184=1015.730,146.640,-133.126,-24.372,21.404,-41.422
C04185=1015.738,146.226,-133.087,-24.372,21.404,-41.424
C04186=1015.745,145.813,-133.048,-24.371,21.405,-41.427
C04187=1015.751,145.401,-133.009,-24.371,21.404,-41.431
C04188=1015.758,144.989,-132.969,-24.370,21.405,-41.432
C04189=1015.764,144.578,-132.930,-24.370,21.405,-41.436
C04190=1015.772,144.167,-132.891,-24.370,21.405,-41.438
C04191=1015.778,143.756,-132.852,-24.369,21.406,-41.442
C04192=1015.785,143.347,-132.813,-24.369,21.405,-41.445
C04193=1015.792,142.939,-132.775,-24.368,21.406,-41.448
C04194=1015.798,142.530,-132.735,-24.368,21.406,-41.451
C04195=1015.805,142.123,-132.697,-24.368,21.406,-41.453
C04196=1015.812,141.717,-132.658,-24.367,21.407,-41.457
C04197=1015.818,141.312,-132.620,-24.366,21.406,-41.460
C04198=1015.825,140.907,-132.581,-24.366,21.407,-41.462
C04199=1015.831,140.490,-132.541,-24.366,21.408,-41.466
C04200=1015.836,140.254,-132.519,-24.366,21.408,-41.468
C04201=1015.839,139.995,-132.494,-24.365,21.408,-41.470
C04202=1015.844,139.719,-132.468,-24.365,21.408,-41.471
C04203=1015.848,139.431,-132.440,-24.365,21.408,-41.473
C04204=1015.853,139.143,-132.414,-24.364,21.408,-41.475
C04205=1015.857,138.865,-132.387,-24.364,21.407,-41.476
C04206=1015.862,138.606,-132.362,-24.364,21.408,-41.478
C04207=1015.865,138.369,-132.340,-24.364,21.408,-41.480
C04208=1015.869,138.151,-132.320,-24.363,21.408,-41.482
C04209=1015.872,137.946,-132.300,-24.363,21.408,-41.484
C04210=1015.878,137.545,-132.262,-24.363,21.408,-41.486
C04211=1015.884,137.175,-132.227,-24.363,21.410,-41.488
C04212=1015.889,136.838,-132.195,-24.362,21.409,-41.491
C04213=1015.895,136.522,-132.164,-24.361,21.409,-41.495
C04214=1015.899,136.205,-132.135,-24.361,21.410,-41.497
C04215=1015.905,135.865,-132.102,-24.361,21.409,-41.500
C04216=1015.910,135.493,-132.067,-24.360,21.410,-41.502
C04217=1015.917,135.098,-132.029,-24.360,21.411,-41.505
C04218=1015.923,134.699,-131.991,-24.360,21.410,-41.508
C04219=1015.929,134.301,-131.954,-24.359,21.411,-41.510
C04220=1015.934,133.902,-131.916,-24.359,21.411,-41.514
C04221=1015.941,133.503,-131.878,-24.358,21.411,-41.517
C04222=1015.947,133.105,-131.840,-24.358,21.412,-41.519
C04223=1015.953,132.706,-131.803,-24.358,21.411,-41.523
C04224=1015.959,132.307,-131.765,-24.357,21.412,-41.525
C04225=1015.965,131.909,-131.726,-24.357,21.412,-41.528
C04226=1015.970,131.511,-131.689,-24.356,21.412,-41.532
C04227=1015.977,131.112,-131.651,-24.356,21.413,-41.534
C04228=1015.983,130.713,-131.613,-24.356,21.413,-41.538
C04229=1015.988,130.315,-131.576,-24.355,21.413,-41.541
C04230=1015.994,129.916,-131.538,-24.355,21.413,-41.543
C04231=1016.000,129.517,-131.500,-24.354,21.413,-41.547
C04232=1016.006,129.119,-131.463,-24.354,21.413,-41.550
C04233=1016.012,128.720,-131.425,-24.354,21.414,-41.552
C04234=1016.018,128.322,-131.386,-24.353,21.414,-41.555
C04235=1016.023,127.924,-131.349,-24.353,21.415,-41.558
C04236=1016.030,127.525,-131.311,-24.352,21.414,-41.561
C04237=1016.035,127.126,-131.274,-24.352,21.415,-41.565
C04238=1016.041,126.728,-131.236,-24.351,21.415,-41.567
C04239=1016.047,126.329,-131.199,-24.351,21.415,-41.571
C04240=1016.053,125.930,-131.161,-24.350,21.415,-41.574
C04241=1016.058,125.533,-131.123,-24.350,21.416,-41.576
C04242=1016.063,125.133,-131.084,-24.350,21.416,-41.580
C04243=1016.069,124.735,-131.047,-24.349,21.416,-41.583
C04244=1016.074,124.336,-131.010,-24.349,21.416,-41.585
C04245=1016.081,123.938,-130.972,-24.348,21.417,-41.589
C04246=1016.086,123.539,-130.935,-24.348,21.416,-41.592
C04247=1016.092,123.141,-130.896,-24.348,21.418,-41.595
C04248=1016.097,122.743,-130.859,-24.347,21.417,-41.598
C04249=1016.103,122.344,-130.821,-24.347,21.418,-41.602
C04250=1016.108,121.946,-130.784,-24.346,21.417,-41.605
C04251=1016.114,121.546,-130.746,-24.346,21.418,-41.607
C04252=1016.119,121.149,-130.708,-24.345,21.418,-41.611
C04253=1016.124,120.750,-130.671,-24.345,21.418,-41.614
C04254=1016.130,120.351,-130.633,-24.345,21.419,-41.617
C04255=1016.136,119.953,-130.595,-24.344,21.419,-41.620
C04256=1016.141,119.555,-130.558,-24.343,21.419,-41.624
C04257=1016.148,119.156,-130.521,-24.343,21.420,-41.626
C04258=1016.154,118.758,-130.483,-24.343,21.420,-41.629
C04259=1016.159,118.360,-130.446,-24.342,21.420,-41.633
C04260=1016.164,117.961,-130.409,-24.342,21.420,-41.637
C04261=1016.171,117.562,-130.372,-24.341,21.420,-41.638
C04262=1016.176,117.163,-130.334,-24.341,21.421,-41.642
C04263=1016.182,116.765,-130.297,-24.340,21.420,-41.646
C04264=1016.187,116.367,-130.260,-24.340,21.421,-41.649
C04265=1016.193,115.968,-130.222,-24.340,21.422,-41.652
C04266=1016.199,115.569,-130.185,-24.339,21.422,-41.655
C04267=1016.205,115.172,-130.148,-24.339,21.422,-41.659
C04268=1016.210,114.773,-130.110,-24.338,21.422,-41.662
C04269=1016.216,114.375,-130.073,-24.338,21.423,-41.664
C04270=1016.221,113.976,-130.036,-24.337,21.422,-41.668
C04271=1016.227,113.578,-129.998,-24.337,21.423,-41.671
C04272=1016.232,113.180,-129.961,-24.336,21.423,-41.675
C04273=1016.237,112.781,-129.924,-24.336,21.423,-41.677
C04274=1016.243,112.383,-129.887,-24.335,21.424,-41.681
C04275=1016.248,111.984,-129.849,-24.335,21.423,-41.684
C04276=1016.254,111.585,-129.813,-24.334,21.424,-41.688
C04277=1016.259,111.186,-129.775,-24.334,21.425,-41.690
C04278=1016.264,110.788,-129.738,-24.334,21.425,-41.694
C04279=1016.270,110.389,-129.700,-24.333,21.425,-41.697
C04280=1016.275,109.991,-129.663,-24.333,21.425,-41.701
C04281=1016.281,109.592,-129.626,-24.332,21.426,-41.703
C04282=1016.286,109.194,-129.589,-24.332,21.426,-41.707
C04283=1016.291,108.795,-129.551,-24.331,21.426,-41.710
C04284=1016.296,108.397,-129.515,-24.331,21.426,-41.714
C04285=1016.301,107.998,-129.477,-24.330,21.426,-41.717
C04286=1016.306,107.600,-129.440,-24.330,21.427,-41.719
C04287=1016.312,107.201,-129.402,-24.330,21.427,-41.723
C04288=1016.318,106.802,-129.366,-24.329,21.427,-41.727
C04289=1016.323,106.404,-129.328,-24.328,21.427,-41.730
C04290=1016.327,106.005,-129.291,-24.328,21.428,-41.734
C04291=1016.333,105.607,-129.254,-24.328,21.428,-41.736
C04292=1016.338,105.208,-129.217,-24.327,21.429,-41.740
C04293=1016.343,104.810,-129.180,-24.327,21.429,-41.743
C04294=1016.348,104.411,-129.142,-24.326,21.429,-41.747
C04295=1016.353,104.013,-129.105,-24.326,21.429,-41.751
C04296=1016.359,103.613,-129.069,-24.325,21.430,-41.754
C04297=1016.363,103.215,-129.032,-24.325,21.430,-41.756
C04298=1016.368,102.816,-128.994,-24.324,21.430,-41.760
C04299=1016.374,102.418,-128.957,-24.324,21.430,-41.763
C04300=1016.378,102.019,-128.920,-24.323,21.430,-41.767
C04301=1016.383,101.621,-128.883,-24.323,21.431,-41.771
C04302=1016.388,101.221,-128.845,-24.322,21.431,-41.775
C04303=1016.393,100.823,-128.809,-24.322,21.431,-41.778
C04304=1016.398,100.424,-128.771,-24.322,21.432,-41.780
C04305=1016.403,100.025,-128.735,-24.321,21.432,-41.784
C04306=1016.407,99.626,-128.697,-24.320,21.432,-41.787
C04307=1016.412,99.228,-128.660,-24.320,21.432,-41.791
C04308=1016.417,98.828,-128.623,-24.319,21.433,-41.795
C04309=1016.422,98.430,-128.587,-24.319,21.432,-41.798
C04310=1016.427,98.031,-128.549,-24.318,21.433,-41.802
C04311=1016.431,97.633,-128.512,-24.318,21.433,-41.806
C04312=1016.437,97.233,-128.475,-24.318,21.434,-41.808
C04313=1016.441,96.834,-128.438,-24.317,21.434,-41.811
C04314=1016.446,96.436,-128.401,-24.317,21.435,-41.815
C04315=1016.450,96.037,-128.364,-24.316,21.435,-41.819
C04316=1016.455,95.637,-128.327,-24.316,21.435,-41.822
C04317=1016.460,95.239,-128.290,-24.315,21.435,-41.826
C04318=1016.464,94.840,-128.253,-24.315,21.436,-41.830
C04319=1016.469,94.441,-128.216,-24.314,21.435,-41.833
C04320=1016.473,94.042,-128.179,-24.313,21.436,-41.837
C04321=1016.478,93.644,-128.142,-24.313,21.436,-41.841
C04322=1016.483,93.244,-128.106,-24.312,21.437,-41.844
C04323=1016.487,92.845,-128.068,-24.312,21.437,-41.846
C04324=1016.491,92.446,-128.031,-24.312,21.437,-41.850
C04325=1016.497,92.047,-127.994,-24.311,21.438,-41.854
C04326=1016.501,91.648,-127.957,-24.311,21.438,-41.857
C04327=1016.505,91.249,-127.920,-24.310,21.438,-41.861
C04328=1016.510,90.849,-127.883,-24.310,21.438,-41.865
C04329=1016.515,90.451,-127.847,-24.309,21.439,-41.868
C04330=1016.519,90.052,-127.810,-24.309,21.439,-41.872
C04331=1016.523,89.653,-127.773,-24.308,21.439,-41.875
C04332=1016.528,89.260,-127.737,-24.308,21.439,-41.879
C04333=1016.531,88.874,-127.701,-24.307,21.440,-41.883
C04334=1016.536,88.491,-127.666,-24.307,21.440,-41.887
C04335=1016.540,88.108,-127.630,-24.306,21.440,-41.890
C04336=1016.544,87.719,-127.595,-24.305,21.440,-41.894
C04337=1016.548,87.323,-127.558,-24.305,21.441,-41.898
C04338=1016.553,86.921,-127.521,-24.304,21.441,-41.901
C04339=1016.558,86.515,-127.483,-24.304,21.442,-41.905
C04340=1016.561,86.107,-127.445,-24.303,21.441,-41.908
C04341=1016.566,85.698,-127.408,-24.303,21.442,-41.912
C04342=1016.571,85.288,-127.370,-24.302,21.442,-41.916
C04343=1016.575,84.876,-127.332,-24.302,21.443,-41.920
C04344=1016.579,84.461,-127.294,-24.301,21.443,-41.923
C04345=1016.583,84.045,-127.256,-24.301,21.443,-41.927
C04346=1016.588,83.628,-127.218,-24.300,21.444,-41.931
C04347=1016.592,83.209,-127.179,-24.300,21.444,-41.935
C04348=1016.596,82.788,-127.140,-24.299,21.444,-41.938
C04349=1016.601,82.367,-127.102,-24.299,21.444,-41.942
C04350=1016.603,82.157,-127.082,-24.299,21.445,-41.944
C04351=1016.605,81.945,-127.062,-24.298,21.444,-41.947
C04352=1016.607,81.733,-127.043,-24.298,21.445,-41.949
C04353=1016.609,81.521,-127.024,-24.298,21.445,-41.951
C04354=1016.611,81.309,-127.005,-24.297,21.445,-41.953
C04355=1016.614,81.096,-126.985,-24.297,21.445,-41.955
C04356=1016.616,80.884,-126.965,-24.297,21.445,-41.956
C04357=1016.617,80.671,-126.946,-24.297,21.446,-41.958
C04358=1016.620,80.458,-126.926,-24.296,21.446,-41.960
C04359=1016.622,80.246,-126.906,-24.296,21.446,-41.962
C04360=1016.624,80.033,-126.887,-24.296,21.446,-41.964
C04361=1016.627,79.823,-126.868,-24.296,21.447,-41.966
C04362=1016.630,79.409,-126.830,-24.295,21.447,-41.970
C04363=1016.634,79.003,-126.793,-24.294,21.447,-41.973
C04364=1016.638,78.607,-126.756,-24.294,21.447,-41.977
C04365=1016.643,78.216,-126.720,-24.293,21.448,-41.980
C04366=1016.646,77.829,-126.684,-24.293,21.447,-41.986
C04367=1016.650,77.444,-126.650,-24.292,21.448,-41.989
C04368=1016.654,77.054,-126.614,-24.292,21.449,-41.994
C04369=1016.658,76.661,-126.577,-24.291,21.449,-41.997
C04370=1016.661,76.258,-126.541,-24.291,21.449,-42.001
C04371=1016.665,75.847,-126.503,-24.290,21.450,-42.004
C04372=1016.669,75.427,-126.464,-24.290,21.450,-42.008
C04373=1016.671,75.214,-126.446,-24.289,21.451,-42.010
C04374=1016.673,75.001,-126.426,-24.289,21.451,-42.012
C04375=1016.675,74.787,-126.407,-24.289,21.450,-42.015
C04376=1016.677,74.574,-126.386,-24.288,21.451,-42.017
C04377=1016.679,74.361,-126.368,-24.288,21.451,-42.019
C04378=1016.681,74.148,-126.348,-24.288,21.451,-42.021
C04379=1016.683,73.936,-126.329,-24.288,21.451,-42.023
C04380=1016.685,73.724,-126.309,-24.287,21.452,-42.025
C04381=1016.689,73.304,-126.271,-24.287,21.452,-42.028
C04382=1016.693,72.886,-126.233,-24.286,21.452,-42.034
C04383=1016.696,72.471,-126.195,-24.285,21.452,-42.037
C04384=1016.700,72.057,-126.157,-24.285,21.453,-42.041
C04385=1016.704,71.645,-126.120,-24.285,21.453,-42.045
C04386=1016.708,71.234,-126.082,-24.284,21.454,-42.049
C04387=1016.712,70.823,-126.044,-24.283,21.453,-42.054
C04388=1016.716,70.412,-126.007,-24.283,21.454,-42.058
C04389=1016.719,70.000,-125.969,-24.282,21.454,-42.061
C04390=1016.722,69.590,-125.932,-24.282,21.455,-42.065
C04391=1016.726,69.180,-125.895,-24.281,21.455,-42.069
C04392=1016.730,68.770,-125.857,-24.280,21.455,-42.074
C04393=1016.733,68.364,-125.820,-24.280,21.456,-42.078
C04394=1016.737,67.958,-125.783,-24.279,21.456,-42.082
C04395=1016.740,67.553,-125.746,-24.279,21.457,-42.085
C04396=1016.744,67.150,-125.710,-24.278,21.457,-42.089
C04397=1016.747,66.747,-125.673,-24.278,21.457,-42.094
C04398=1016.751,66.347,-125.637,-24.277,21.457,-42.098
C04399=1016.754,65.948,-125.600,-24.277,21.458,-42.102
C04400=1016.757,65.541,-125.563,-24.276,21.458,-42.106
C04401=1016.760,65.328,-125.545,-24.276,21.459,-42.108
C04402=1016.761,65.106,-125.525,-24.275,21.458,-42.111
C04403=1016.764,64.876,-125.503,-24.275,21.458,-42.113
C04404=1016.765,64.640,-125.482,-24.275,21.459,-42.115
C04405=1016.767,64.405,-125.460,-24.274,21.459,-42.116
C04406=1016.769,64.175,-125.440,-24.274,21.459,-42.120
C04407=1016.771,63.958,-125.420,-24.274,21.460,-42.122
C04408=1016.772,63.750,-125.401,-24.274,21.460,-42.124
C04409=1016.774,63.533,-125.382,-24.273,21.459,-42.127
C04410=1016.776,63.284,-125.359,-24.273,21.460,-42.129
C04411=1016.779,63.016,-125.334,-24.272,21.460,-42.131
C04412=1016.780,62.762,-125.311,-24.272,21.460,-42.133
C04413=1016.784,62.350,-125.275,-24.271,21.461,-42.139
C04414=1016.787,61.956,-125.239,-24.271,21.461,-42.142
C04415=1016.790,61.542,-125.201,-24.270,21.462,-42.146
C04416=1016.793,61.142,-125.165,-24.270,21.462,-42.150
C04417=1016.796,60.742,-125.129,-24.269,21.462,-42.155
C04418=1016.800,60.342,-125.092,-24.269,21.463,-42.159
C04419=1016.803,59.942,-125.057,-24.268,21.463,-42.163
C04420=1016.806,59.541,-125.020,-24.268,21.464,-42.166
C04421=1016.809,59.141,-124.984,-24.267,21.463,-42.172
C04422=1016.812,58.742,-124.948,-24.266,21.464,-42.175
C04423=1016.815,58.342,-124.912,-24.266,21.464,-42.179
C04424=1016.819,57.941,-124.876,-24.265,21.465,-42.183
C04425=1016.822,57.540,-124.840,-24.264,21.465,-42.188
C04426=1016.825,57.140,-124.803,-24.264,21.465,-42.192
C04427=1016.828,56.741,-124.767,-24.264,21.466,-42.196
C04428=1016.831,56.340,-124.732,-24.263,21.465,-42.201
C04429=1016.834,55.940,-124.695,-24.262,21.467,-42.205
C04430=1016.837,55.540,-124.659,-24.262,21.467,-42.209
C04431=1016.840,55.140,-124.623,-24.261,21.468,-42.212
C04432=1016.842,54.739,-124.588,-24.260,21.468,-42.218
C04433=1016.845,54.339,-124.552,-24.260,21.468,-42.221
C04434=1016.848,53.939,-124.516,-24.259,21.468,-42.225
C04435=1016.851,53.540,-124.480,-24.259,21.468,-42.230
C04436=1016.854,53.138,-124.444,-24.258,21.469,-42.234
C04437=1016.857,52.738,-124.408,-24.258,21.469,-42.238
C04438=1016.860,52.339,-124.372,-24.257,21.469,-42.243
C04439=1016.862,51.938,-124.336,-24.256,21.470,-42.247
C04440=1016.865,51.538,-124.300,-24.256,21.471,-42.251
C04441=1016.868,51.138,-124.264,-24.255,21.471,-42.255
C04442=1016.870,50.739,-124.229,-24.255,21.471,-42.260
C04443=1016.873,50.338,-124.192,-24.254,21.472,-42.264
C04444=1016.876,49.937,-124.157,-24.254,21.472,-42.268
C04445=1016.879,49.538,-124.121,-24.253,21.472,-42.273
C04446=1016.881,49.137,-124.085,-24.252,21.473,-42.277
C04447=1016.884,48.737,-124.049,-24.251,21.472,-42.282
C04448=1016.887,48.337,-124.014,-24.251,21.474,-42.286
C04449=1016.889,47.937,-123.977,-24.251,21.474,-42.290
C04450=1016.891,47.537,-123.942,-24.250,21.474,-42.295
C04451=1016.895,47.137,-123.906,-24.249,21.475,-42.299
C04452=1016.897,46.737,-123.871,-24.249,21.475,-42.302
C04453=1016.900,46.337,-123.834,-24.248,21.475,-42.308
C04454=1016.902,45.937,-123.800,-24.247,21.475,-42.311
C04455=1016.905,45.536,-123.763,-24.247,21.477,-42.316
C04456=1016.907,45.136,-123.728,-24.246,21.477,-42.321
C04457=1016.910,44.736,-123.693,-24.246,21.477,-42.325
C04458=1016.913,44.336,-123.657,-24.245,21.477,-42.330
C04459=1016.915,43.936,-123.621,-24.244,21.477,-42.333
C04460=1016.917,43.537,-123.585,-24.244,21.479,-42.338
C04461=1016.920,43.136,-123.550,-24.243,21.479,-42.343
C04462=1016.922,42.736,-123.514,-24.243,21.479,-42.347
C04463=1016.924,42.336,-123.478,-24.242,21.479,-42.352
C04464=1016.927,41.936,-123.444,-24.241,21.479,-42.356
C04465=1016.929,41.536,-123.408,-24.241,21.480,-42.359
C04466=1016.931,41.137,-123.372,-24.240,21.481,-42.365
C04467=1016.934,40.737,-123.336,-24.240,21.481,-42.369
C04468=1016.937,40.337,-123.301,-24.239,21.481,-42.374
C04469=1016.938,39.936,-123.265,-24.238,21.481,-42.378
C04470=1016.941,39.537,-123.230,-24.238,21.482,-42.383
C04471=1016.943,39.137,-123.195,-24.237,21.483,-42.387
C04472=1016.946,38.737,-123.159,-24.237,21.483,-42.391
C04473=1016.947,38.337,-123.124,-24.236,21.483,-42.396
C04474=1016.950,37.937,-123.088,-24.235,21.483,-42.400
C04475=1016.952,37.537,-123.053,-24.235,21.484,-42.405
C04476=1016.954,37.138,-123.018,-24.234,21.485,-42.409
C04477=1016.956,36.738,-122.982,-24.233,21.484,-42.414
C04478=1016.958,36.338,-122.948,-24.233,21.485,-42.418
C04479=1016.961,35.938,-122.912,-24.232,21.486,-42.424
C04480=1016.963,35.538,-122.877,-24.231,21.486,-42.428
C04481=1016.965,35.139,-122.842,-24.231,21.486,-42.433
C04482=1016.967,34.738,-122.806,-24.230,21.486,-42.437
C04483=1016.969,34.339,-122.771,-24.229,21.487,-42.442
C04484=1016.970,33.940,-122.736,-24.229,21.488,-42.446
C04485=1016.973,33.540,-122.701,-24.228,21.487,-42.451
C04486=1016.975,33.140,-122.666,-24.228,21.489,-42.455
C04487=1016.976,32.740,-122.630,-24.227,21.489,-42.461
C04488=1016.979,32.340,-122.595,-24.226,21.489,-42.464
C04489=1016.980,31.941,-122.560,-24.226,21.489,-42.469
C04490=1016.983,31.541,-122.525,-24.225,21.490,-42.474
C04491=1016.985,31.142,-122.490,-24.224,21.490,-42.479
C04492=1016.987,30.742,-122.455,-24.224,21.491,-42.483
C04493=1016.988,30.343,-122.420,-24.223,21.491,-42.488
C04494=1016.991,29.944,-122.384,-24.223,21.492,-42.492
C04495=1016.992,29.543,-122.350,-24.222,21.492,-42.497
C04496=1016.994,29.144,-122.315,-24.221,21.492,-42.501
C04497=1016.995,28.745,-122.280,-24.221,21.493,-42.507
C04498=1016.998,28.345,-122.244,-24.220,21.493,-42.510
C04499=1016.999,27.945,-122.210,-24.219,21.493,-42.516
C04500=1017.001,27.546,-122.175,-24.219,21.495,-42.520
C04501=1017.003,27.147,-122.140,-24.218,21.494,-42.525
C04502=1017.005,26.747,-122.105,-24.218,21.495,-42.529
C04503=1017.007,26.348,-122.070,-24.217,21.496,-42.534
C04504=1017.008,25.949,-122.035,-24.216,21.496,-42.540
C04505=1017.010,25.549,-122.001,-24.215,21.496,-42.543
C04506=1017.012,25.150,-121.966,-24.215,21.497,-42.549
C04507=1017.013,24.751,-121.931,-24.214,21.497,-42.553
C04508=1017.015,24.351,-121.896,-24.213,21.497,-42.558
C04509=1017.016,23.968,-121.862,-24.213,21.498,-42.562
C04510=1017.017,23.638,-121.834,-24.213,21.498,-42.564
C04511=1017.019,23.366,-121.810,-24.212,21.498,-42.567
C04512=1017.020,23.132,-121.790,-24.211,21.499,-42.573
C04513=1017.021,22.900,-121.769,-24.211,21.500,-42.577
C04514=1017.022,22.634,-121.747,-24.211,21.500,-42.580
C04515=1017.022,22.312,-121.718,-24.210,21.500,-42.584
C04516=1017.025,21.937,-121.686,-24.210,21.501,-42.586
C04517=1017.026,21.524,-121.650,-24.209,21.501,-42.593
C04518=1017.027,21.279,-121.629,-24.208,21.501,-42.597
C04519=1017.028,21.007,-121.606,-24.208,21.502,-42.599
C04520=1017.029,20.716,-121.580,-24.207,21.501,-42.602
C04521=1017.030,20.419,-121.554,-24.207,21.501,-42.604
C04522=1017.031,20.132,-121.530,-24.207,21.503,-42.606
C04523=1017.032,19.866,-121.506,-24.206,21.502,-42.610
C04524=1017.032,19.629,-121.486,-24.206,21.503,-42.613
C04525=1017.033,19.418,-121.468,-24.205,21.503,-42.617
C04526=1017.035,19.021,-121.433,-24.205,21.503,-42.622
C04527=1017.037,18.624,-121.399,-24.204,21.503,-42.626
C04528=1017.038,18.229,-121.365,-24.203,21.504,-42.632
C04529=1017.040,17.834,-121.331,-24.203,21.505,-42.635
C04530=1017.040,17.439,-121.296,-24.202,21.505,-42.641
C04531=1017.042,17.047,-121.263,-24.201,21.505,-42.646
C04532=1017.042,16.654,-121.228,-24.201,21.506,-42.650
C04533=1017.045,16.262,-121.195,-24.200,21.506,-42.656
C04534=1017.046,15.871,-121.161,-24.200,21.507,-42.659
C04535=1017.047,15.481,-121.127,-24.199,21.507,-42.665
C04536=1017.049,15.091,-121.093,-24.198,21.508,-42.670
C04537=1017.050,14.702,-121.061,-24.198,21.508,-42.674
C04538=1017.050,14.314,-121.028,-24.197,21.509,-42.680
C04539=1017.052,13.926,-120.993,-24.196,21.509,-42.683
C04540=1017.053,13.539,-120.960,-24.196,21.509,-42.689
C04541=1017.054,13.152,-120.927,-24.195,21.511,-42.693
C04542=1017.055,12.765,-120.893,-24.194,21.510,-42.698
C04543=1017.056,12.380,-120.861,-24.193,21.510,-42.703
C04544=1017.057,11.992,-120.828,-24.193,21.512,-42.707
C04545=1017.059,11.606,-120.794,-24.192,21.511,-42.713
C04546=1017.060,11.221,-120.761,-24.192,21.512,-42.716
C04547=1017.060,10.838,-120.728,-24.191,21.513,-42.722
C04548=1017.061,10.457,-120.696,-24.191,21.513,-42.726
C04549=1017.063,10.078,-120.663,-24.190,21.513,-42.731
C04550=1017.063,9.703,-120.631,-24.189,21.514,-42.737
C04551=1017.064,9.327,-120.599,-24.189,21.514,-42.740
C04552=1017.066,8.950,-120.567,-24.188,21.515,-42.746
C04553=1017.066,8.572,-120.534,-24.187,21.515,-42.751
C04554=1017.067,8.191,-120.502,-24.187,21.516,-42.755
C04555=1017.068,7.807,-120.469,-24.186,21.516,-42.761
C04556=1017.069,7.420,-120.436,-24.185,21.517,-42.764
C04557=1017.069,7.029,-120.403,-24.185,21.517,-42.770
C04558=1017.070,6.636,-120.370,-24.184,21.517,-42.775
C04559=1017.072,6.244,-120.336,-24.183,21.519,-42.779
C04560=1017.072,5.850,-120.302,-24.182,21.518,-42.785
C04561=1017.073,5.455,-120.269,-24.182,21.519,-42.790
C04562=1017.074,5.060,-120.235,-24.181,21.520,-42.794
C04563=1017.075,4.665,-120.201,-24.180,21.519,-42.799
C04564=1017.076,4.269,-120.168,-24.180,21.520,-42.805
C04565=1017.076,3.880,-120.134,-24.179,21.521,-42.809
C04566=1017.077,3.521,-120.104,-24.179,21.521,-42.812
C04567=1017.077,3.193,-120.076,-24.178,21.521,-42.817
C04568=1017.078,2.879,-120.050,-24.177,21.522,-42.823
C04569=1017.079,2.557,-120.022,-24.177,21.522,-42.827
C04570=1017.080,2.203,-119.993,-24.176,21.523,-42.833
C04571=1017.080,1.818,-119.960,-24.175,21.524,-42.836
C04572=1017.080,1.420,-119.926,-24.175,21.523,-42.841
C04573=1017.081,1.022,-119.892,-24.174,21.525,-42.846
C04574=1017.082,0.621,-119.858,-24.173,21.525,-42.851
C04575=1017.082,0.220,-119.825,-24.173,21.525,-42.857
C04576=1017.083,-0.183,-119.791,-24.172,21.525,-42.862
C04577=1017.083,-0.589,-119.756,-24.171,21.526,-42.867
C04578=1017.084,-0.998,-119.722,-24.171,21.527,-42.872
C04579=1017.084,-1.408,-119.688,-24.170,21.527,-42.877
C04580=1017.085,-1.820,-119.652,-24.169,21.528,-42.882
C04581=1017.085,-2.235,-119.617,-24.169,21.529,-42.888
C04582=1017.086,-2.652,-119.582,-24.168,21.529,-42.893
C04583=1017.087,-3.071,-119.547,-24.167,21.529,-42.899
C04584=1017.087,-3.493,-119.512,-24.166,21.530,-42.904
C04585=1017.087,-3.704,-119.493,-24.166,21.530,-42.908
C04586=1017.087,-3.917,-119.476,-24.165,21.530,-42.910
C04587=1017.088,-4.130,-119.458,-24.165,21.530,-42.913
C04588=1017.088,-4.346,-119.439,-24.165,21.531,-42.915
C04589=1017.088,-4.562,-119.422,-24.164,21.531,-42.919
C04590=1017.088,-4.781,-119.403,-24.164,21.531,-42.921
C04591=1017.089,-5.001,-119.385,-24.163,21.532,-42.925
C04592=1017.089,-5.222,-119.366,-24.163,21.532,-42.927
C04593=1017.089,-5.444,-119.348,-24.163,21.532,-42.930
C04594=1017.089,-5.668,-119.329,-24.162,21.532,-42.934
C04595=1017.089,-5.892,-119.310,-24.162,21.533,-42.935
C04596=1017.089,-6.117,-119.292,-24.161,21.533,-42.939
C04597=1017.089,-6.340,-119.273,-24.161,21.533,-42.941
C04598=1017.090,-6.564,-119.254,-24.161,21.533,-42.944
C04599=1017.090,-6.788,-119.235,-24.160,21.534,-42.947
C04600=1017.090,-7.010,-119.216,-24.160,21.534,-42.950
C04601=1017.091,-7.232,-119.198,-24.160,21.535,-42.952
C04602=1017.090,-7.452,-119.180,-24.159,21.534,-42.956
C04603=1017.091,-7.671,-119.162,-24.159,21.535,-42.959
C04604=1017.091,-7.889,-119.144,-24.158,21.535,-42.961
C04605=1017.091,-8.106,-119.125,-24.158,21.536,-42.965
C04606=1017.091,-8.323,-119.107,-24.158,21.536,-42.967
C04607=1017.091,-8.540,-119.089,-24.157,21.536,-42.971
C04608=1017.091,-8.757,-119.070,-24.157,21.537,-42.973
C04609=1017.091,-8.974,-119.052,-24.156,21.536,-42.976
C04610=1017.092,-9.190,-119.035,-24.156,21.537,-42.980
C04611=1017.091,-9.406,-119.016,-24.156,21.537,-42.982
C04612=1017.092,-9.622,-118.999,-24.155,21.538,-42.985
C04613=1017.092,-9.839,-118.981,-24.155,21.538,-42.987
C04614=1017.092,-10.054,-118.962,-24.154,21.538,-42.991
C04615=1017.092,-10.270,-118.945,-24.154,21.539,-42.993
C04616=1017.092,-10.486,-118.926,-24.154,21.538,-42.996
C04617=1017.092,-10.700,-118.909,-24.153,21.539,-42.998
C04618=1017.092,-10.916,-118.890,-24.153,21.539,-43.002
C04619=1017.092,-11.130,-118.873,-24.152,21.539,-43.006
C04620=1017.092,-11.343,-118.855,-24.152,21.540,-43.007
C04621=1017.092,-11.557,-118.837,-24.152,21.540,-43.011
C04622=1017.093,-11.769,-118.820,-24.151,21.540,-43.013
C04623=1017.092,-11.982,-118.802,-24.151,21.540,-43.016
C04624=1017.093,-12.193,-118.784,-24.151,21.541,-43.019
C04625=1017.092,-12.405,-118.767,-24.150,21.541,-43.022
C04626=1017.092,-12.616,-118.749,-24.150,21.542,-43.024
C04627=1017.092,-13.035,-118.714,-24.149,21.542,-43.029
C04628=1017.092,-13.452,-118.680,-24.148,21.543,-43.035
C04629=1017.092,-13.868,-118.645,-24.148,21.543,-43.041
C04630=1017.092,-14.279,-118.612,-24.147,21.544,-43.046
C04631=1017.092,-14.687,-118.578,-24.146,21.544,-43.052
C04632=1017.092,-15.092,-118.544,-24.145,21.545,-43.057
C04633=1017.092,-15.495,-118.511,-24.145,21.545,-43.063
C04634=1017.092,-15.897,-118.477,-24.144,21.546,-43.068
C04635=1017.092,-16.296,-118.444,-24.143,21.546,-43.074
C04636=1017.091,-16.694,-118.411,-24.142,21.547,-43.079
C04637=1017.092,-17.092,-118.379,-24.142,21.548,-43.085
C04638=1017.091,-17.491,-118.346,-24.141,21.547,-43.090
C04639=1017.091,-17.901,-118.312,-24.140,21.548,-43.098
C04640=1017.090,-18.149,-118.292,-24.139,21.549,-43.101
C04641=1017.091,-18.437,-118.268,-24.139,21.549,-43.105
C04642=1017.091,-18.748,-118.243,-24.139,21.550,-43.107
C04643=1017.090,-19.060,-118.217,-24.139,21.550,-43.109
C04644=1017.090,-19.347,-118.193,-24.138,21.550,-43.113
C04645=1017.090,-19.596,-118.173,-24.138,21.551,-43.116
C04646=1017.089,-20.008,-118.139,-24.136,21.551,-43.123
C04647=1017.089,-20.406,-118.106,-24.136,21.552,-43.129
C04648=1017.088,-20.803,-118.074,-24.135,21.553,-43.135
C04649=1017.088,-21.201,-118.041,-24.134,21.552,-43.140
C04650=1017.088,-21.598,-118.008,-24.134,21.553,-43.146
C04651=1017.088,-21.995,-117.976,-24.133,21.554,-43.151
C04652=1017.087,-22.394,-117.943,-24.132,21.554,-43.156
C04653=1017.086,-22.791,-117.911,-24.131,21.555,-43.162
C04654=1017.086,-23.188,-117.878,-24.131,21.555,-43.168
C04655=1017.085,-23.586,-117.846,-24.130,21.556,-43.173
C04656=1017.085,-23.983,-117.813,-24.129,21.556,-43.178
C04657=1017.085,-24.381,-117.781,-24.128,21.557,-43.184
C04658=1017.085,-24.778,-117.748,-24.128,21.558,-43.190
C04659=1017.084,-25.175,-117.716,-24.127,21.558,-43.195
C04660=1017.082,-25.573,-117.683,-24.126,21.558,-43.201
C04661=1017.082,-25.971,-117.651,-24.125,21.559,-43.206
C04662=1017.082,-26.368,-117.618,-24.125,21.560,-43.212
C04663=1017.081,-26.765,-117.586,-24.124,21.560,-43.217
C04664=1017.080,-27.163,-117.554,-24.123,21.561,-43.221
C04665=1017.080,-27.560,-117.521,-24.123,21.562,-43.227
C04666=1017.079,-27.957,-117.489,-24.122,21.562,-43.232
C04667=1017.078,-28.356,-117.457,-24.121,21.562,-43.238
C04668=1017.078,-28.753,-117.425,-24.120,21.563,-43.243
C04669=1017.077,-29.150,-117.393,-24.120,21.564,-43.249
C04670=1017.076,-29.548,-117.361,-24.119,21.565,-43.255
C04671=1017.075,-29.945,-117.328,-24.118,21.565,-43.260
C04672=1017.074,-30.342,-117.296,-24.117,21.565,-43.265
C04673=1017.073,-30.740,-117.264,-24.117,21.566,-43.271
C04674=1017.072,-31.137,-117.232,-24.116,21.567,-43.277
C04675=1017.072,-31.535,-117.199,-24.115,21.568,-43.282
C04676=1017.071,-31.932,-117.168,-24.114,21.567,-43.287
C04677=1017.070,-32.330,-117.136,-24.114,21.568,-43.293
C04678=1017.070,-32.727,-117.104,-24.113,21.569,-43.299
C04679=1017.068,-33.125,-117.071,-24.112,21.570,-43.304
C04680=1017.067,-33.522,-117.039,-24.111,21.570,-43.310
C04681=1017.066,-33.919,-117.007,-24.111,21.570,-43.315
C04682=1017.065,-34.317,-116.976,-24.110,21.571,-43.321
C04683=1017.065,-34.714,-116.944,-24.109,21.571,-43.328
C04684=1017.063,-35.111,-116.912,-24.108,21.572,-43.334
C04685=1017.062,-35.509,-116.879,-24.107,21.572,-43.339
C04686=1017.061,-35.906,-116.847,-24.107,21.573,-43.344
C04687=1017.059,-36.303,-116.816,-24.106,21.573,-43.350
C04688=1017.059,-36.701,-116.784,-24.105,21.574,-43.356
C04689=1017.057,-37.098,-116.753,-24.105,21.575,-43.361
C04690=1017.056,-37.496,-116.720,-24.104,21.575,-43.366
C04691=1017.055,-37.893,-116.688,-24.103,21.576,-43.372
C04692=1017.054,-38.290,-116.656,-24.102,21.576,-43.378
C04693=1017.053,-38.688,-116.625,-24.102,21.577,-43.383
C04694=1017.052,-39.085,-116.593,-24.101,21.578,-43.389
C04695=1017.050,-39.482,-116.562,-24.100,21.578,-43.394
C04696=1017.049,-39.880,-116.529,-24.099,21.579,-43.400
C04697=1017.047,-40.277,-116.497,-24.099,21.579,-43.405
C04698=1017.046,-40.674,-116.467,-24.098,21.580,-43.411
C04699=1017.045,-41.071,-116.435,-24.097,21.581,-43.417
C04700=1017.044,-41.468,-116.403,-24.096,21.582,-43.422
C04701=1017.042,-41.866,-116.371,-24.096,21.582,-43.427
C04702=1017.041,-42.264,-116.340,-24.095,21.582,-43.433
C04703=1017.039,-42.661,-116.308,-24.094,21.583,-43.439
C04704=1017.038,-43.057,-116.277,-24.093,21.584,-43.444
C04705=1017.036,-43.454,-116.245,-24.092,21.584,-43.451
C04706=1017.035,-43.852,-116.214,-24.092,21.585,-43.457
C04707=1017.033,-44.250,-116.182,-24.091,21.585,-43.462
C04708=1017.031,-44.647,-116.151,-24.090,21.585,-43.468
C04709=1017.030,-45.043,-116.119,-24.089,21.586,-43.473
C04710=1017.029,-45.441,-116.088,-24.089,21.587,-43.479
C04711=1017.027,-45.838,-116.057,-24.088,21.588,-43.485
C04712=1017.025,-46.236,-116.025,-24.087,21.589,-43.490
C04713=1017.023,-46.632,-115.993,-24.086,21.588,-43.496
C04714=1017.022,-47.030,-115.962,-24.086,21.589,-43.501
C04715=1017.021,-47.427,-115.931,-24.085,21.590,-43.507
C04716=1017.019,-47.824,-115.900,-24.084,21.591,-43.512
C04717=1017.017,-48.220,-115.868,-24.084,21.592,-43.518
C04718=1017.015,-48.619,-115.837,-24.083,21.592,-43.525
C04719=1017.013,-49.015,-115.806,-24.082,21.592,-43.531
C04720=1017.011,-49.412,-115.774,-24.081,21.592,-43.536
C04721=1017.010,-49.809,-115.743,-24.080,21.593,-43.542
C04722=1017.008,-50.206,-115.712,-24.080,21.594,-43.547
C04723=1017.007,-50.603,-115.681,-24.079,21.595,-43.553
C04724=1017.004,-51.000,-115.650,-24.078,21.595,-43.558
C04725=1017.003,-51.397,-115.618,-24.077,21.596,-43.564
C04726=1017.000,-51.795,-115.588,-24.077,21.597,-43.570
C04727=1016.998,-52.191,-115.557,-24.076,21.598,-43.575
C04728=1016.996,-52.588,-115.525,-24.075,21.598,-43.581
C04729=1016.994,-52.985,-115.494,-24.074,21.598,-43.588
C04730=1016.992,-53.382,-115.463,-24.073,21.599,-43.593
C04731=1016.991,-53.779,-115.432,-24.073,21.599,-43.599
C04732=1016.988,-54.176,-115.401,-24.072,21.600,-43.604
C04733=1016.986,-54.572,-115.370,-24.071,21.601,-43.610
C04734=1016.984,-54.970,-115.340,-24.071,21.602,-43.616
C04735=1016.982,-55.367,-115.308,-24.070,21.603,-43.621
C04736=1016.980,-55.764,-115.277,-24.069,21.602,-43.627
C04737=1016.977,-56.162,-115.246,-24.068,21.603,-43.632
C04738=1016.976,-56.559,-115.215,-24.067,21.603,-43.639
C04739=1016.974,-56.957,-115.185,-24.067,21.604,-43.645
C04740=1016.971,-57.356,-115.153,-24.066,21.605,-43.651
C04741=1016.969,-57.780,-115.121,-24.065,21.606,-43.656
C04742=1016.967,-58.154,-115.092,-24.064,21.606,-43.662
C04743=1016.965,-58.553,-115.061,-24.064,21.607,-43.667
C04744=1016.962,-58.954,-115.030,-24.063,21.608,-43.673
C04745=1016.959,-59.354,-114.998,-24.062,21.608,-43.680
C04746=1016.957,-59.756,-114.967,-24.061,21.609,-43.686
C04747=1016.955,-60.157,-114.936,-24.061,21.610,-43.691
C04748=1016.952,-60.560,-114.905,-24.060,21.610,-43.697
C04749=1016.950,-60.963,-114.874,-24.059,21.610,-43.702
C04750=1016.947,-61.367,-114.843,-24.058,21.611,-43.708
C04751=1016.944,-61.770,-114.812,-24.057,21.611,-43.715
C04752=1016.942,-62.175,-114.780,-24.057,21.612,-43.720
C04753=1016.939,-62.581,-114.749,-24.056,21.613,-43.726
C04754=1016.936,-62.987,-114.718,-24.055,21.614,-43.732
C04755=1016.934,-63.393,-114.686,-24.054,21.615,-43.737
C04756=1016.931,-63.799,-114.655,-24.053,21.615,-43.744
C04757=1016.929,-64.206,-114.624,-24.053,21.615,-43.750
C04758=1016.926,-64.615,-114.592,-24.052,21.616,-43.756
C04759=1016.923,-65.022,-114.561,-24.051,21.617,-43.761
C04760=1016.921,-65.431,-114.530,-24.050,21.617,-43.768
C04761=1016.918,-65.840,-114.498,-24.049,21.618,-43.774
C04762=1016.915,-66.249,-114.467,-24.049,21.619,-43.780
C04763=1016.912,-66.658,-114.436,-24.048,21.620,-43.785
C04764=1016.909,-67.068,-114.404,-24.047,21.620,-43.791
C04765=1016.906,-67.478,-114.373,-24.046,21.621,-43.798
C04766=1016.903,-67.889,-114.341,-24.046,21.621,-43.804
C04767=1016.900,-68.299,-114.310,-24.045,21.622,-43.809
C04768=1016.897,-68.709,-114.278,-24.044,21.623,-43.815
C04769=1016.894,-69.120,-114.248,-24.043,21.623,-43.822
C04770=1016.891,-69.531,-114.216,-24.042,21.624,-43.827
C04771=1016.888,-69.942,-114.185,-24.042,21.625,-43.833
C04772=1016.884,-70.353,-114.153,-24.041,21.625,-43.839
C04773=1016.883,-70.764,-114.122,-24.040,21.626,-43.846
C04774=1016.879,-71.174,-114.090,-24.039,21.626,-43.851
C04775=1016.876,-71.586,-114.060,-24.039,21.627,-43.857
C04776=1016.873,-71.997,-114.028,-24.038,21.628,-43.865
C04777=1016.869,-72.408,-113.997,-24.037,21.629,-43.870
C04778=1016.865,-72.818,-113.966,-24.036,21.630,-43.876
C04779=1016.862,-73.229,-113.934,-24.035,21.631,-43.881
C04780=1016.859,-73.640,-113.903,-24.034,21.631,-43.888
C04781=1016.856,-74.050,-113.872,-24.034,21.632,-43.894
C04782=1016.852,-74.461,-113.841,-24.033,21.632,-43.900
C04783=1016.849,-74.871,-113.810,-24.032,21.633,-43.905
C04784=1016.846,-75.281,-113.779,-24.031,21.633,-43.912
C04785=1016.842,-75.692,-113.748,-24.031,21.634,-43.918
C04786=1016.839,-76.100,-113.717,-24.030,21.635,-43.924
C04787=1016.835,-76.510,-113.686,-24.029,21.636,-43.929
C04788=1016.832,-76.919,-113.654,-24.028,21.636,-43.936
C04789=1016.828,-77.328,-113.625,-24.027,21.637,-43.942
C04790=1016.825,-77.736,-113.594,-24.027,21.637,-43.948
C04791=1016.821,-78.144,-113.563,-24.026,21.638,-43.953
C04792=1016.817,-78.552,-113.531,-24.025,21.638,-43.960
C04793=1016.814,-78.959,-113.501,-24.024,21.639,-43.966
C04794=1016.810,-79.366,-113.470,-24.023,21.640,-43.972
C04795=1016.806,-79.771,-113.441,-24.023,21.641,-43.977
C04796=1016.803,-80.177,-113.409,-24.022,21.641,-43.984
C04797=1016.799,-80.582,-113.380,-24.021,21.642,-43.990
C04798=1016.795,-80.987,-113.349,-24.020,21.643,-43.995
C04799=1016.791,-81.391,-113.318,-24.020,21.643,-44.001
C04800=1016.787,-81.794,-113.288,-24.019,21.644,-44.007
C04801=1016.783,-82.197,-113.257,-24.018,21.644,-44.014
C04802=1016.780,-82.599,-113.228,-24.017,21.645,-44.019
C04803=1016.776,-83.001,-113.197,-24.016,21.646,-44.025
C04804=1016.772,-83.401,-113.168,-24.016,21.647,-44.031
C04805=1016.767,-83.802,-113.138,-24.015,21.648,-44.036
C04806=1016.765,-84.202,-113.108,-24.014,21.648,-44.043
C04807=1016.760,-84.608,-113.078,-24.013,21.649,-44.049
C04808=1016.758,-84.832,-113.061,-24.013,21.649,-44.053
C04809=1016.756,-85.072,-113.043,-24.012,21.650,-44.056
C04810=1016.753,-85.326,-113.024,-24.012,21.649,-44.060
C04811=1016.750,-85.580,-113.005,-24.012,21.650,-44.062
C04812=1016.748,-85.827,-112.987,-24.011,21.650,-44.065
C04813=1016.745,-86.057,-112.969,-24.011,21.651,-44.069
C04814=1016.741,-86.466,-112.939,-24.010,21.652,-44.077
C04815=1016.737,-86.854,-112.910,-24.009,21.652,-44.082
C04816=1016.733,-87.234,-112.881,-24.008,21.652,-44.087
C04817=1016.730,-87.606,-112.854,-24.007,21.653,-44.093
C04818=1016.726,-87.977,-112.826,-24.007,21.654,-44.099
C04819=1016.722,-88.353,-112.799,-24.006,21.655,-44.104
C04820=1016.717,-88.760,-112.768,-24.005,21.656,-44.112
C04821=1016.715,-89.008,-112.750,-24.005,21.656,-44.116
C04822=1016.711,-89.282,-112.729,-24.004,21.657,-44.117
C04823=1016.708,-89.567,-112.709,-24.004,21.656,-44.121
C04824=1016.706,-89.842,-112.688,-24.003,21.657,-44.124
C04825=1016.703,-90.091,-112.669,-24.003,21.657,-44.128
C04826=1016.701,-90.310,-112.653,-24.002,21.658,-44.132
C04827=1016.695,-90.707,-112.623,-24.002,21.659,-44.138
C04828=1016.691,-91.100,-112.595,-24.001,21.659,-44.145
C04829=1016.687,-91.493,-112.565,-24.000,21.660,-44.150
C04830=1016.682,-91.885,-112.537,-23.999,21.660,-44.156
C04831=1016.678,-92.276,-112.508,-23.999,21.661,-44.162
C04832=1016.674,-92.667,-112.479,-23.998,21.662,-44.167
C04833=1016.670,-93.057,-112.450,-23.997,21.663,-44.173
C04834=1016.665,-93.446,-112.421,-23.996,21.664,-44.178
C04835=1016.660,-93.835,-112.393,-23.996,21.664,-44.184
C04836=1016.656,-94.222,-112.364,-23.995,21.664,-44.189
C04837=1016.651,-94.609,-112.335,-23.994,21.665,-44.195
C04838=1016.647,-94.996,-112.307,-23.994,21.666,-44.200
C04839=1016.643,-95.381,-112.279,-23.993,21.666,-44.207
C04840=1016.638,-95.766,-112.250,-23.992,21.667,-44.213
C04841=1016.634,-96.151,-112.222,-23.991,21.668,-44.219
C04842=1016.628,-96.535,-112.194,-23.990,21.668,-44.224
C04843=1016.624,-96.918,-112.165,-23.990,21.669,-44.230
C04844=1016.619,-97.302,-112.137,-23.989,21.669,-44.235
C04845=1016.615,-97.685,-112.109,-23.988,21.670,-44.241
C04846=1016.610,-98.068,-112.081,-23.988,21.671,-44.246
C04847=1016.605,-98.452,-112.053,-23.987,21.672,-44.252
C04848=1016.600,-98.835,-112.025,-23.986,21.673,-44.258
C04849=1016.596,-99.219,-111.996,-23.985,21.673,-44.263
C04850=1016.590,-99.603,-111.968,-23.985,21.673,-44.268
C04851=1016.585,-99.987,-111.940,-23.984,21.674,-44.274
C04852=1016.580,-100.372,-111.912,-23.983,21.675,-44.280
C04853=1016.576,-100.757,-111.883,-23.982,21.676,-44.285
C04854=1016.570,-101.142,-111.855,-23.982,21.677,-44.291
C04855=1016.566,-101.528,-111.827,-23.981,21.676,-44.296
C04856=1016.561,-101.915,-111.799,-23.980,21.677,-44.302
C04857=1016.555,-102.304,-111.771,-23.980,21.678,-44.307
C04858=1016.550,-102.692,-111.743,-23.979,21.678,-44.314
C04859=1016.545,-103.081,-111.714,-23.978,21.679,-44.320
C04860=1016.540,-103.471,-111.686,-23.977,21.680,-44.326
C04861=1016.534,-103.862,-111.658,-23.976,21.681,-44.331
C04862=1016.529,-104.253,-111.628,-23.976,21.682,-44.337
C04863=1016.524,-104.644,-111.600,-23.975,21.681,-44.342
C04864=1016.518,-105.036,-111.572,-23.974,21.682,-44.348
C04865=1016.513,-105.429,-111.543,-23.974,21.683,-44.353
C04866=1016.508,-105.821,-111.515,-23.973,21.684,-44.359
C04867=1016.502,-106.214,-111.486,-23.972,21.685,-44.365
C04868=1016.497,-106.607,-111.457,-23.971,21.686,-44.370
C04869=1016.491,-107.000,-111.429,-23.971,21.686,-44.376
C04870=1016.486,-107.393,-111.400,-23.970,21.687,-44.383
C04871=1016.480,-107.786,-111.371,-23.969,21.687,-44.388
C04872=1016.475,-108.179,-111.343,-23.968,21.688,-44.394
C04873=1016.469,-108.572,-111.314,-23.968,21.688,-44.399
C04874=1016.463,-108.965,-111.285,-23.967,21.689,-44.405
C04875=1016.457,-109.358,-111.258,-23.966,21.690,-44.411
C04876=1016.451,-109.750,-111.229,-23.965,21.691,-44.416
C04877=1016.446,-110.144,-111.201,-23.965,21.691,-44.422
C04878=1016.440,-110.536,-111.173,-23.964,21.692,-44.427
C04879=1016.434,-110.929,-111.143,-23.963,21.693,-44.433
C04880=1016.428,-111.322,-111.116,-23.963,21.694,-44.439
C04881=1016.422,-111.715,-111.087,-23.962,21.694,-44.446
C04882=1016.416,-112.107,-111.059,-23.961,21.694,-44.451
C04883=1016.410,-112.500,-111.030,-23.960,21.695,-44.456
C04884=1016.404,-112.893,-111.002,-23.959,21.696,-44.462
C04885=1016.398,-113.286,-110.973,-23.959,21.696,-44.468
C04886=1016.392,-113.678,-110.945,-23.958,21.697,-44.473
C04887=1016.385,-114.071,-110.917,-23.957,21.698,-44.479
C04888=1016.379,-114.463,-110.888,-23.957,21.699,-44.485
C04889=1016.374,-114.856,-110.860,-23.956,21.700,-44.490
C04890=1016.367,-115.248,-110.832,-23.955,21.701,-44.496
C04891=1016.361,-115.641,-110.804,-23.954,21.700,-44.501
C04892=1016.355,-116.033,-110.775,-23.954,21.701,-44.507
C04893=1016.349,-116.425,-110.747,-23.953,21.702,-44.512
C04894=1016.342,-116.818,-110.719,-23.952,21.703,-44.518
C04895=1016.336,-117.210,-110.691,-23.952,21.704,-44.523
C04896=1016.329,-117.603,-110.662,-23.951,21.705,-44.529
C04897=1016.323,-117.995,-110.634,-23.950,21.705,-44.536
C04898=1016.316,-118.387,-110.606,-23.949,21.705,-44.541
C04899=1016.309,-118.779,-110.578,-23.948,21.706,-44.547
C04900=1016.303,-119.172,-110.550,-23.948,21.706,-44.553
C04901=1016.297,-119.564,-110.521,-23.947,21.707,-44.558
C04902=1016.289,-119.956,-110.494,-23.946,21.708,-44.564
C04903=1016.283,-120.348,-110.465,-23.946,21.709,-44.569
C04904=1016.276,-120.741,-110.437,-23.945,21.710,-44.575
C04905=1016.270,-121.133,-110.409,-23.944,21.710,-44.580
C04906=1016.263,-121.526,-110.381,-23.943,21.710,-44.586
C04907=1016.256,-121.917,-110.353,-23.943,21.711,-44.591
C04908=1016.249,-122.310,-110.325,-23.942,21.712,-44.597
C04909=1016.242,-122.701,-110.297,-23.941,21.713,-44.603
C04910=1016.235,-123.094,-110.269,-23.941,21.714,-44.608
C04911=1016.229,-123.486,-110.241,-23.940,21.715,-44.614
C04912=1016.221,-123.878,-110.213,-23.939,21.714,-44.619
C04913=1016.214,-124.270,-110.185,-23.939,21.715,-44.625
C04914=1016.208,-124.663,-110.157,-23.938,21.716,-44.630
C04915=1016.200,-125.054,-110.128,-23.937,21.717,-44.636
C04916=1016.193,-125.446,-110.101,-23.936,21.718,-44.642
C04917=1016.186,-125.839,-110.073,-23.936,21.719,-44.647
C04918=1016.179,-126.230,-110.045,-23.935,21.719,-44.652
C04919=1016.171,-126.622,-110.017,-23.934,21.719,-44.658
C04920=1016.164,-127.015,-109.989,-23.934,21.720,-44.664
C04921=1016.157,-127.406,-109.961,-23.933,21.721,-44.669
C04922=1016.149,-127.798,-109.933,-23.932,21.722,-44.675
C04923=1016.142,-128.191,-109.905,-23.932,21.723,-44.680
C04924=1016.135,-128.582,-109.877,-23.931,21.723,-44.686
C04925=1016.127,-128.974,-109.848,-23.930,21.723,-44.691
C04926=1016.119,-129.366,-109.821,-23.929,21.724,-44.697
C04927=1016.112,-129.758,-109.794,-23.929,21.725,-44.703
C04928=1016.104,-130.150,-109.765,-23.928,21.726,-44.708
C04929=1016.097,-130.542,-109.737,-23.927,21.727,-44.714
C04930=1016.089,-130.933,-109.710,-23.926,21.727,-44.719
C04931=1016.081,-131.325,-109.682,-23.926,21.728,-44.725
C04932=1016.073,-131.717,-109.654,-23.925,21.728,-44.730
C04933=1016.066,-132.109,-109.626,-23.924,21.729,-44.736
C04934=1016.057,-132.501,-109.598,-23.924,21.730,-44.741
C04935=1016.050,-132.892,-109.570,-23.923,21.730,-44.747
C04936=1016.042,-133.285,-109.543,-23.922,21.731,-44.752
C04937=1016.034,-133.676,-109.514,-23.922,21.732,-44.758
C04938=1016.026,-134.068,-109.487,-23.921,21.732,-44.763
C04939=1016.428,-134.039,-109.737,-23.921,21.732,-44.763
C04940=1016.435,-133.648,-109.765,-23.922,21.732,-44.758
C04941=1016.444,-133.255,-109.793,-23.922,21.731,-44.752
C04942=1016.450,-132.864,-109.820,-23.923,21.730,-44.747
C04943=1016.459,-132.472,-109.848,-23.924,21.730,-44.741
C04944=1016.466,-132.080,-109.876,-23.924,21.729,-44.736
C04945=1016.474,-131.688,-109.903,-23.925,21.728,-44.730
C04946=1016.481,-131.297,-109.931,-23.926,21.728,-44.725
C04947=1016.488,-130.904,-109.959,-23.926,21.727,-44.719
C04948=1016.495,-130.513,-109.987,-23.927,21.727,-44.714
C04949=1016.504,-130.121,-110.014,-23.928,21.726,-44.708
C04950=1016.510,-129.729,-110.042,-23.929,21.725,-44.703
C04951=1016.518,-129.337,-110.070,-23.929,21.724,-44.697
C04952=1016.525,-128.945,-110.097,-23.930,21.723,-44.691
C04953=1016.532,-128.553,-110.125,-23.931,21.723,-44.686
C04954=1016.539,-128.162,-110.153,-23.932,21.723,-44.680
C04955=1016.546,-127.770,-110.181,-23.932,21.722,-44.675
C04956=1016.554,-127.377,-110.209,-23.933,21.721,-44.669
C04957=1016.560,-126.986,-110.236,-23.934,21.720,-44.664
C04958=1016.568,-126.593,-110.264,-23.934,21.719,-44.658
C04959=1016.575,-126.202,-110.292,-23.935,21.719,-44.652
C04960=1016.582,-125.810,-110.319,-23.936,21.719,-44.647
C04961=1016.589,-125.417,-110.347,-23.936,21.718,-44.642
C04962=1016.595,-125.025,-110.375,-23.937,21.717,-44.636
C04963=1016.602,-124.634,-110.403,-23.938,21.716,-44.630
C04964=1016.609,-124.241,-110.431,-23.939,21.715,-44.625
C04965=1016.615,-123.849,-110.459,-23.939,21.714,-44.619
C04966=1016.622,-123.457,-110.486,-23.940,21.715,-44.614
C04967=1016.630,-123.065,-110.514,-23.941,21.714,-44.608
C04968=1016.636,-122.673,-110.542,-23.941,21.713,-44.603
C04969=1016.643,-122.281,-110.570,-23.942,21.712,-44.597
C04970=1016.649,-121.889,-110.598,-23.943,21.711,-44.591
C04971=1016.656,-121.497,-110.626,-23.943,21.710,-44.586
C04972=1016.662,-121.105,-110.654,-23.944,21.710,-44.580
C04973=1016.669,-120.712,-110.682,-23.945,21.710,-44.575
C04974=1016.676,-120.320,-110.710,-23.946,21.709,-44.569
C04975=1016.682,-119.928,-110.738,-23.946,21.708,-44.564
C04976=1016.689,-119.536,-110.766,-23.947,21.707,-44.558
C04977=1016.695,-119.143,-110.795,-23.948,21.706,-44.553
C04978=1016.702,-118.752,-110.822,-23.948,21.706,-44.547
C04979=1016.707,-118.359,-110.850,-23.949,21.705,-44.541
C04980=1016.714,-117.966,-110.878,-23.950,21.705,-44.536
C04981=1016.720,-117.574,-110.906,-23.951,21.705,-44.529
C04982=1016.726,-117.182,-110.934,-23.952,21.704,-44.523
C04983=1016.733,-116.790,-110.963,-23.952,21.703,-44.518
C04984=1016.739,-116.397,-110.990,-23.953,21.702,-44.512
C04985=1016.745,-116.005,-111.018,-23.954,21.701,-44.507
C04986=1016.750,-115.612,-111.047,-23.954,21.700,-44.501
C04987=1016.757,-115.220,-111.075,-23.955,21.701,-44.496
C04988=1016.763,-114.827,-111.103,-23.956,21.700,-44.490
C04989=1016.769,-114.435,-111.131,-23.957,21.699,-44.485
C04990=1016.776,-114.042,-111.160,-23.957,21.698,-44.479
C04991=1016.781,-113.649,-111.188,-23.958,21.697,-44.473
C04992=1016.787,-113.257,-111.216,-23.959,21.696,-44.468
C04993=1016.792,-112.865,-111.244,-23.959,21.696,-44.462
C04994=1016.798,-112.472,-111.272,-23.960,21.695,-44.456
C04995=1016.805,-112.079,-111.300,-23.961,21.694,-44.451
C04996=1016.810,-111.687,-111.329,-23.962,21.694,-44.446
C04997=1016.816,-111.293,-111.357,-23.963,21.694,-44.439
C04998=1016.822,-110.901,-111.385,-23.963,21.693,-44.433
C04999=1016.827,-110.508,-111.413,-23.964,21.692,-44.427
C05000=1016.833,-110.115,-111.443,-23.965,21.691,-44.422
C05001=1016.838,-109.723,-111.470,-23.965,21.691,-44.416
C05002=1016.844,-109.330,-111.499,-23.966,21.690,-44.411
C05003=1016.849,-108.937,-111.527,-23.967,21.689,-44.405
C05004=1016.855,-108.544,-111.556,-23.968,21.688,-44.399
C05005=1016.861,-108.151,-111.584,-23.968,21.688,-44.394
C05006=1016.866,-107.758,-111.613,-23.969,21.687,-44.388
C05007=1016.872,-107.366,-111.640,-23.970,21.687,-44.383
C05008=1016.877,-106.972,-111.669,-23.971,21.686,-44.376
C05009=1016.882,-106.579,-111.698,-23.971,21.686,-44.370
C05010=1016.887,-106.186,-111.726,-23.972,21.685,-44.365
C05011=1016.893,-105.793,-111.755,-23.973,21.684,-44.359
C05012=1016.898,-105.400,-111.783,-23.974,21.683,-44.353
C05013=1016.903,-105.008,-111.812,-23.974,21.682,-44.348
C05014=1016.909,-104.617,-111.839,-23.975,21.681,-44.342
C05015=1016.914,-104.225,-111.868,-23.976,21.682,-44.337
C05016=1016.919,-103.834,-111.897,-23.976,21.681,-44.331
C05017=1016.925,-103.443,-111.925,-23.977,21.680,-44.326
C05018=1016.930,-103.053,-111.953,-23.978,21.679,-44.320
C05019=1016.935,-102.665,-111.982,-23.979,21.678,-44.314
C05020=1016.940,-102.276,-112.010,-23.980,21.678,-44.307
C05021=1016.944,-101.888,-112.038,-23.980,21.677,-44.302
C05022=1016.949,-101.501,-112.067,-23.981,21.676,-44.296
C05023=1016.954,-101.115,-112.094,-23.982,21.677,-44.291
C05024=1016.959,-100.729,-112.123,-23.982,21.676,-44.285
C05025=1016.963,-100.343,-112.151,-23.983,21.675,-44.280
C05026=1016.969,-99.959,-112.179,-23.984,21.674,-44.274
C05027=1016.973,-99.555,-112.208,-23.985,21.673,-44.268
C05028=1016.978,-99.172,-112.236,-23.985,21.673,-44.263
C05029=1016.982,-98.808,-112.264,-23.986,21.673,-44.258
C05030=1016.987,-98.424,-112.291,-23.987,21.672,-44.252
C05031=1016.992,-98.041,-112.319,-23.988,21.671,-44.246
C05032=1016.997,-97.658,-112.347,-23.988,21.670,-44.241
C05033=1017.001,-97.274,-112.376,-23.989,21.669,-44.235
C05034=1017.006,-96.890,-112.403,-23.990,21.669,-44.230
C05035=1017.010,-96.507,-112.432,-23.990,21.668,-44.224
C05036=1017.015,-96.123,-112.460,-23.991,21.668,-44.219
C05037=1017.020,-95.738,-112.488,-23.992,21.667,-44.213
C05038=1017.024,-95.353,-112.516,-23.993,21.666,-44.207
C05039=1017.028,-94.968,-112.545,-23.994,21.666,-44.200
C05040=1017.033,-94.582,-112.573,-23.994,21.665,-44.195
C05041=1017.037,-94.195,-112.601,-23.995,21.664,-44.189
C05042=1017.042,-93.807,-112.630,-23.996,21.664,-44.184
C05043=1017.045,-93.419,-112.659,-23.996,21.664,-44.178
C05044=1017.050,-93.030,-112.687,-23.997,21.663,-44.173
C05045=1017.055,-92.640,-112.716,-23.998,21.662,-44.167
C05046=1017.058,-92.249,-112.745,-23.999,21.661,-44.162
C05047=1017.063,-91.858,-112.774,-23.999,21.660,-44.156
C05048=1017.067,-91.466,-112.803,-24.000,21.660,-44.150
C05049=1017.072,-91.073,-112.831,-24.001,21.659,-44.145
C05050=1017.075,-90.679,-112.860,-24.002,21.659,-44.138
C05051=1017.080,-90.283,-112.890,-24.002,21.658,-44.132
C05052=1017.083,-90.064,-112.906,-24.003,21.657,-44.128
C05053=1017.085,-89.814,-112.924,-24.003,21.657,-44.124
C05054=1017.088,-89.539,-112.945,-24.004,21.656,-44.121
C05055=1017.091,-89.255,-112.966,-24.004,21.657,-44.117
C05056=1017.094,-88.981,-112.986,-24.005,21.656,-44.116
C05057=1017.096,-88.734,-113.005,-24.005,21.656,-44.112
C05058=1017.100,-88.326,-113.035,-24.006,21.655,-44.104
C05059=1017.105,-87.950,-113.062,-24.007,21.654,-44.099
C05060=1017.108,-87.578,-113.090,-24.007,21.653,-44.093
C05061=1017.111,-87.206,-113.118,-24.008,21.652,-44.087
C05062=1017.116,-86.827,-113.146,-24.009,21.652,-44.082
C05063=1017.120,-86.439,-113.175,-24.010,21.652,-44.077
C05064=1017.124,-86.029,-113.205,-24.011,21.651,-44.069
C05065=1017.126,-85.800,-113.222,-24.011,21.650,-44.065
C05066=1017.129,-85.553,-113.241,-24.012,21.650,-44.062
C05067=1017.131,-85.298,-113.260,-24.012,21.649,-44.060
C05068=1017.134,-85.045,-113.278,-24.012,21.650,-44.056
C05069=1017.136,-84.804,-113.297,-24.013,21.649,-44.053
C05070=1017.138,-84.581,-113.313,-24.013,21.649,-44.049
C05071=1017.142,-84.174,-113.344,-24.014,21.648,-44.043
C05072=1017.146,-83.774,-113.373,-24.015,21.648,-44.036
C05073=1017.150,-83.374,-113.403,-24.016,21.647,-44.031
C05074=1017.153,-82.974,-113.433,-24.016,21.646,-44.025
C05075=1017.157,-82.572,-113.463,-24.017,21.645,-44.019
C05076=1017.161,-82.170,-113.494,-24.018,21.644,-44.014
C05077=1017.165,-81.767,-113.524,-24.019,21.644,-44.007
C05078=1017.168,-81.363,-113.553,-24.020,21.643,-44.001
C05079=1017.172,-80.960,-113.584,-24.020,21.643,-43.995
C05080=1017.175,-80.555,-113.615,-24.021,21.642,-43.990
C05081=1017.179,-80.150,-113.644,-24.022,21.641,-43.984
C05082=1017.183,-79.745,-113.675,-24.023,21.641,-43.977
C05083=1017.186,-79.339,-113.705,-24.023,21.640,-43.972
C05084=1017.190,-78.931,-113.736,-24.024,21.639,-43.966
C05085=1017.194,-78.525,-113.766,-24.025,21.638,-43.960
C05086=1017.197,-78.116,-113.797,-24.026,21.638,-43.953
C05087=1017.200,-77.709,-113.828,-24.027,21.637,-43.948
C05088=1017.204,-77.300,-113.859,-24.027,21.637,-43.942
C05089=1017.208,-76.892,-113.889,-24.028,21.636,-43.936
C05090=1017.211,-76.483,-113.920,-24.029,21.636,-43.929
C05091=1017.214,-76.074,-113.952,-24.030,21.635,-43.924
C05092=1017.218,-75.664,-113.983,-24.031,21.634,-43.918
C05093=1017.221,-75.254,-114.013,-24.031,21.633,-43.912
C05094=1017.224,-74.844,-114.045,-24.032,21.633,-43.905
C05095=1017.228,-74.433,-114.075,-24.033,21.632,-43.900
C05096=1017.231,-74.023,-114.106,-24.034,21.632,-43.894
C05097=1017.235,-73.613,-114.137,-24.034,21.631,-43.888
C05098=1017.238,-73.202,-114.168,-24.035,21.631,-43.881
C05099=1017.241,-72.791,-114.200,-24.036,21.630,-43.876
C05100=1017.244,-72.380,-114.231,-24.037,21.629,-43.870
C05101=1017.247,-71.969,-114.262,-24.038,21.628,-43.865
C05102=1017.250,-71.559,-114.293,-24.039,21.627,-43.857
C05103=1017.253,-71.148,-114.325,-24.039,21.626,-43.851
C05104=1017.257,-70.737,-114.356,-24.040,21.626,-43.846
C05105=1017.260,-70.325,-114.387,-24.041,21.625,-43.839
C05106=1017.263,-69.915,-114.418,-24.042,21.625,-43.833
C05107=1017.266,-69.504,-114.449,-24.042,21.624,-43.827
C05108=1017.269,-69.093,-114.481,-24.043,21.623,-43.822
C05109=1017.272,-68.682,-114.513,-24.044,21.623,-43.815
C05110=1017.274,-68.271,-114.543,-24.045,21.622,-43.809
C05111=1017.277,-67.861,-114.575,-24.046,21.621,-43.804
C05112=1017.280,-67.451,-114.606,-24.046,21.621,-43.798
C05113=1017.283,-67.041,-114.638,-24.047,21.620,-43.791
C05114=1017.285,-66.631,-114.669,-24.048,21.620,-43.785
C05115=1017.289,-66.222,-114.701,-24.049,21.619,-43.780
C05116=1017.292,-65.813,-114.731,-24.049,21.618,-43.774
C05117=1017.294,-65.404,-114.763,-24.050,21.617,-43.768
C05118=1017.297,-64.996,-114.794,-24.051,21.617,-43.761
C05119=1017.300,-64.587,-114.826,-24.052,21.616,-43.756
C05120=1017.303,-64.180,-114.856,-24.053,21.615,-43.750
C05121=1017.305,-63.772,-114.888,-24.053,21.615,-43.744
C05122=1017.308,-63.365,-114.920,-24.054,21.615,-43.737
C05123=1017.310,-62.959,-114.951,-24.055,21.614,-43.732
C05124=1017.313,-62.553,-114.982,-24.056,21.613,-43.726
C05125=1017.316,-62.149,-115.013,-24.057,21.612,-43.720
C05126=1017.318,-61.744,-115.045,-24.057,21.611,-43.715
C05127=1017.320,-61.340,-115.075,-24.058,21.611,-43.708
C05128=1017.323,-60.936,-115.107,-24.059,21.610,-43.702
C05129=1017.325,-60.533,-115.137,-24.060,21.610,-43.697
C05130=1017.328,-60.131,-115.169,-24.061,21.610,-43.691
C05131=1017.329,-59.729,-115.200,-24.061,21.609,-43.686
C05132=1017.333,-59.328,-115.231,-24.062,21.608,-43.680
C05133=1017.335,-58.927,-115.262,-24.063,21.608,-43.673
C05134=1017.337,-58.527,-115.293,-24.064,21.607,-43.667
C05135=1017.340,-58.127,-115.324,-24.064,21.606,-43.662
C05136=1017.341,-57.728,-115.355,-24.065,21.606,-43.656
C05137=1017.344,-57.329,-115.386,-24.066,21.605,-43.651
C05138=1017.346,-56.931,-115.417,-24.067,21.604,-43.645
C05139=1017.348,-56.533,-115.448,-24.067,21.603,-43.639
C05140=1017.350,-56.135,-115.479,-24.068,21.603,-43.632
C05141=1017.352,-55.737,-115.510,-24.069,21.602,-43.627
C05142=1017.355,-55.340,-115.541,-24.070,21.603,-43.621
C05143=1017.356,-54.943,-115.571,-24.071,21.602,-43.616
C05144=1017.359,-54.546,-115.602,-24.071,21.601,-43.610
C05145=1017.360,-54.148,-115.633,-24.072,21.600,-43.604
C05146=1017.362,-53.752,-115.664,-24.073,21.599,-43.599
C05147=1017.364,-53.355,-115.695,-24.073,21.599,-43.593
C05148=1017.367,-52.959,-115.726,-24.074,21.598,-43.588
C05149=1017.368,-52.561,-115.757,-24.075,21.598,-43.581
C05150=1017.370,-52.164,-115.788,-24.076,21.598,-43.575
C05151=1017.372,-51.768,-115.820,-24.077,21.597,-43.570
C05152=1017.374,-51.371,-115.851,-24.077,21.596,-43.564
C05153=1017.376,-50.974,-115.881,-24.078,21.595,-43.558
C05154=1017.377,-50.577,-115.912,-24.079,21.595,-43.553
C05155=1017.380,-50.179,-115.944,-24.080,21.594,-43.547
C05156=1017.382,-49.783,-115.975,-24.080,21.593,-43.542
C05157=1017.383,-49.385,-116.006,-24.081,21.592,-43.536
C05158=1017.385,-48.988,-116.037,-24.082,21.592,-43.531
C05159=1017.387,-48.591,-116.069,-24.083,21.592,-43.525
C05160=1017.388,-48.194,-116.100,-24.084,21.592,-43.518
C05161=1017.390,-47.797,-116.131,-24.084,21.591,-43.512
C05162=1017.392,-47.400,-116.162,-24.085,21.590,-43.507
C05163=1017.394,-47.003,-116.194,-24.086,21.589,-43.501
C05164=1017.395,-46.605,-116.225,-24.086,21.588,-43.496
C05165=1017.396,-46.208,-116.257,-24.087,21.589,-43.490
C05166=1017.398,-45.811,-116.288,-24.088,21.588,-43.485
C05167=1017.400,-45.414,-116.319,-24.089,21.587,-43.479
C05168=1017.401,-45.017,-116.350,-24.089,21.586,-43.473
C05169=1017.403,-44.620,-116.382,-24.090,21.585,-43.468
C05170=1017.405,-44.223,-116.414,-24.091,21.585,-43.462
C05171=1017.406,-43.825,-116.445,-24.092,21.585,-43.457
C05172=1017.407,-43.428,-116.477,-24.092,21.584,-43.451
C05173=1017.409,-43.031,-116.508,-24.093,21.584,-43.444
C05174=1017.410,-42.633,-116.539,-24.094,21.583,-43.439
C05175=1017.411,-42.236,-116.571,-24.095,21.582,-43.433
C05176=1017.413,-41.839,-116.602,-24.096,21.582,-43.427
C05177=1017.415,-41.442,-116.634,-24.096,21.582,-43.422
C05178=1017.415,-41.044,-116.666,-24.097,21.581,-43.417
C05179=1017.417,-40.647,-116.697,-24.098,21.580,-43.411
C05180=1017.418,-40.250,-116.729,-24.099,21.579,-43.405
C05181=1017.420,-39.853,-116.761,-24.099,21.579,-43.400
C05182=1017.420,-39.455,-116.792,-24.100,21.578,-43.394
C05183=1017.422,-39.058,-116.824,-24.101,21.578,-43.389
C05184=1017.423,-38.660,-116.856,-24.102,21.577,-43.383
C05185=1017.425,-38.264,-116.888,-24.102,21.576,-43.378
C05186=1017.425,-37.866,-116.920,-24.103,21.576,-43.372
C05187=1017.427,-37.469,-116.951,-24.104,21.575,-43.366
C05188=1017.427,-37.071,-116.983,-24.105,21.575,-43.361
C05189=1017.429,-36.675,-117.015,-24.105,21.574,-43.356
C05190=1017.430,-36.277,-117.047,-24.106,21.573,-43.350
C05191=1017.432,-35.879,-117.078,-24.107,21.573,-43.344
C05192=1017.432,-35.482,-117.110,-24.107,21.572,-43.339
C05193=1017.433,-35.085,-117.142,-24.108,21.572,-43.334
C05194=1017.435,-34.688,-117.174,-24.109,21.571,-43.328
C05195=1017.435,-34.290,-117.206,-24.110,21.571,-43.321
C05196=1017.436,-33.893,-117.238,-24.111,21.570,-43.315
C05197=1017.437,-33.495,-117.270,-24.111,21.570,-43.310
C05198=1017.439,-33.098,-117.302,-24.112,21.570,-43.304
C05199=1017.439,-32.700,-117.334,-24.113,21.569,-43.299
C05200=1017.440,-32.303,-117.366,-24.114,21.568,-43.293
C05201=1017.441,-31.906,-117.398,-24.114,21.567,-43.287
C05202=1017.441,-31.508,-117.430,-24.115,21.568,-43.282
C05203=1017.443,-31.110,-117.462,-24.116,21.567,-43.277
C05204=1017.444,-30.713,-117.495,-24.117,21.566,-43.271
C05205=1017.444,-30.316,-117.527,-24.117,21.565,-43.265
C05206=1017.445,-29.918,-117.559,-24.118,21.565,-43.260
C05207=1017.446,-29.521,-117.591,-24.119,21.565,-43.255
C05208=1017.447,-29.124,-117.623,-24.120,21.564,-43.249
C05209=1017.447,-28.727,-117.655,-24.120,21.563,-43.243
C05210=1017.449,-28.328,-117.687,-24.121,21.562,-43.238
C05211=1017.449,-27.931,-117.720,-24.122,21.562,-43.232
C05212=1017.449,-27.533,-117.752,-24.123,21.562,-43.227
C05213=1017.450,-27.136,-117.784,-24.123,21.561,-43.221
C05214=1017.451,-26.739,-117.817,-24.124,21.560,-43.217
C05215=1017.452,-26.342,-117.849,-24.125,21.560,-43.212
C05216=1017.452,-25.944,-117.882,-24.125,21.559,-43.206
C05217=1017.452,-25.547,-117.914,-24.126,21.558,-43.201
C05218=1017.454,-25.149,-117.946,-24.127,21.558,-43.195
C05219=1017.454,-24.751,-117.979,-24.128,21.558,-43.190
C05220=1017.455,-24.354,-118.011,-24.128,21.557,-43.184
C05221=1017.455,-23.956,-118.044,-24.129,21.556,-43.178
C05222=1017.455,-23.559,-118.076,-24.130,21.556,-43.173
C05223=1017.455,-23.161,-118.108,-24.131,21.555,-43.168
C05224=1017.456,-22.764,-118.140,-24.131,21.555,-43.162
C05225=1017.456,-22.366,-118.173,-24.132,21.554,-43.156
C05226=1017.457,-21.969,-118.205,-24.133,21.554,-43.151
C05227=1017.457,-21.571,-118.239,-24.134,21.553,-43.146
C05228=1017.458,-21.173,-118.271,-24.134,21.552,-43.140
C05229=1017.458,-20.776,-118.304,-24.135,21.553,-43.135
C05230=1017.458,-20.378,-118.336,-24.136,21.552,-43.129
C05231=1017.459,-19.981,-118.369,-24.136,21.551,-43.123
C05232=1017.459,-19.570,-118.403,-24.138,21.551,-43.116
C05233=1017.459,-19.321,-118.423,-24.138,21.550,-43.113
C05234=1017.459,-19.033,-118.447,-24.139,21.550,-43.109
C05235=1017.460,-18.721,-118.472,-24.139,21.550,-43.107
C05236=1017.459,-18.410,-118.498,-24.139,21.549,-43.105
C05237=1017.460,-18.123,-118.522,-24.139,21.549,-43.101
C05238=1017.460,-17.874,-118.543,-24.140,21.548,-43.098
C05239=1017.461,-17.463,-118.576,-24.141,21.547,-43.090
C05240=1017.461,-17.066,-118.609,-24.142,21.548,-43.085
C05241=1017.461,-16.667,-118.642,-24.142,21.547,-43.079
C05242=1017.461,-16.268,-118.675,-24.143,21.546,-43.074
C05243=1017.461,-15.869,-118.707,-24.144,21.546,-43.068
C05244=1017.461,-15.469,-118.742,-24.145,21.545,-43.063
C05245=1017.461,-15.066,-118.775,-24.145,21.545,-43.057
C05246=1017.461,-14.660,-118.808,-24.146,21.544,-43.052
C05247=1017.461,-14.251,-118.842,-24.147,21.544,-43.046
C05248=1017.461,-13.840,-118.876,-24.148,21.543,-43.041
C05249=1017.462,-13.426,-118.910,-24.148,21.543,-43.035
C05250=1017.462,-13.008,-118.945,-24.149,21.542,-43.029
C05251=1017.461,-12.589,-118.979,-24.150,21.542,-43.024
C05252=1017.461,-12.378,-118.997,-24.150,21.541,-43.022
C05253=1017.461,-12.167,-119.015,-24.151,21.541,-43.019
C05254=1017.462,-11.954,-119.032,-24.151,21.540,-43.016
C05255=1017.461,-11.743,-119.050,-24.151,21.540,-43.013
C05256=1017.461,-11.530,-119.068,-24.152,21.540,-43.011
C05257=1017.460,-11.316,-119.085,-24.152,21.540,-43.007
C05258=1017.461,-11.102,-119.103,-24.152,21.539,-43.006
C05259=1017.461,-10.888,-119.121,-24.153,21.539,-43.002
C05260=1017.461,-10.674,-119.138,-24.153,21.539,-42.998
C05261=1017.461,-10.458,-119.157,-24.154,21.538,-42.996
C05262=1017.461,-10.243,-119.175,-24.154,21.539,-42.993
C05263=1017.462,-10.028,-119.193,-24.154,21.538,-42.991
C05264=1017.461,-9.812,-119.210,-24.155,21.538,-42.987
C05265=1017.461,-9.596,-119.228,-24.155,21.538,-42.985
C05266=1017.461,-9.379,-119.246,-24.156,21.537,-42.982
C05267=1017.460,-9.163,-119.264,-24.156,21.537,-42.980
C05268=1017.460,-8.946,-119.283,-24.156,21.536,-42.976
C05269=1017.460,-8.729,-119.301,-24.157,21.537,-42.973
C05270=1017.460,-8.513,-119.318,-24.157,21.536,-42.971
C05271=1017.460,-8.297,-119.336,-24.158,21.536,-42.967
C05272=1017.460,-8.080,-119.355,-24.158,21.536,-42.965
C05273=1017.460,-7.863,-119.373,-24.158,21.535,-42.961
C05274=1017.460,-7.645,-119.391,-24.159,21.535,-42.959
C05275=1017.460,-7.426,-119.410,-24.159,21.534,-42.956
C05276=1017.459,-7.206,-119.429,-24.160,21.535,-42.952
C05277=1017.459,-6.984,-119.447,-24.160,21.534,-42.950
C05278=1017.460,-6.761,-119.466,-24.160,21.534,-42.947
C05279=1017.459,-6.538,-119.484,-24.161,21.533,-42.944
C05280=1017.459,-6.315,-119.503,-24.161,21.533,-42.941
C05281=1017.459,-6.090,-119.521,-24.161,21.533,-42.939
C05282=1017.459,-5.866,-119.540,-24.162,21.533,-42.935
C05283=1017.459,-5.641,-119.559,-24.162,21.532,-42.934
C05284=1017.458,-5.418,-119.578,-24.163,21.532,-42.930
C05285=1017.457,-5.195,-119.596,-24.163,21.532,-42.927
C05286=1017.458,-4.974,-119.616,-24.163,21.532,-42.925
C05287=1017.458,-4.754,-119.633,-24.164,21.531,-42.921
C05288=1017.458,-4.536,-119.652,-24.164,21.531,-42.919
C05289=1017.457,-4.319,-119.670,-24.165,21.531,-42.915
C05290=1017.457,-4.103,-119.689,-24.165,21.530,-42.913
C05291=1017.457,-3.890,-119.706,-24.165,21.530,-42.910
C05292=1017.457,-3.677,-119.724,-24.166,21.530,-42.908
C05293=1017.457,-3.466,-119.742,-24.166,21.530,-42.904
C05294=1017.456,-3.045,-119.778,-24.167,21.529,-42.899
C05295=1017.455,-2.626,-119.813,-24.168,21.529,-42.893
C05296=1017.455,-2.208,-119.848,-24.169,21.529,-42.888
C05297=1017.454,-1.794,-119.882,-24.169,21.528,-42.882
C05298=1017.454,-1.380,-119.917,-24.170,21.527,-42.877
C05299=1017.453,-0.970,-119.952,-24.171,21.527,-42.872
C05300=1017.453,-0.563,-119.986,-24.171,21.526,-42.867
C05301=1017.452,-0.158,-120.021,-24.172,21.525,-42.862
C05302=1017.452,0.246,-120.055,-24.173,21.525,-42.857
C05303=1017.451,0.648,-120.089,-24.173,21.525,-42.851
C05304=1017.450,1.048,-120.123,-24.174,21.525,-42.846
C05305=1017.450,1.446,-120.157,-24.175,21.523,-42.841
C05306=1017.449,1.845,-120.190,-24.175,21.524,-42.836
C05307=1017.448,2.231,-120.223,-24.176,21.523,-42.833
C05308=1017.448,2.583,-120.252,-24.177,21.522,-42.827
C05309=1017.447,2.906,-120.280,-24.177,21.522,-42.823
C05310=1017.447,3.219,-120.306,-24.178,21.521,-42.817
C05311=1017.446,3.547,-120.334,-24.179,21.521,-42.812
C05312=1017.445,3.907,-120.365,-24.179,21.521,-42.809
C05313=1017.444,4.295,-120.398,-24.180,21.520,-42.805
C05314=1017.443,4.691,-120.432,-24.180,21.519,-42.799
C05315=1017.443,5.088,-120.465,-24.181,21.520,-42.794
C05316=1017.443,5.482,-120.499,-24.182,21.519,-42.790
C05317=1017.441,5.877,-120.532,-24.182,21.518,-42.785
C05318=1017.441,6.270,-120.566,-24.183,21.519,-42.779
C05319=1017.440,6.664,-120.599,-24.184,21.517,-42.775
C05320=1017.439,7.056,-120.633,-24.185,21.517,-42.770
C05321=1017.438,7.446,-120.666,-24.185,21.517,-42.764
C05322=1017.437,7.834,-120.699,-24.186,21.516,-42.761
C05323=1017.436,8.218,-120.732,-24.187,21.516,-42.755
C05324=1017.435,8.598,-120.765,-24.187,21.515,-42.751
C05325=1017.434,8.977,-120.797,-24.188,21.515,-42.746
C05326=1017.434,9.353,-120.829,-24.189,21.514,-42.740
C05327=1017.432,9.728,-120.861,-24.189,21.514,-42.737
C05328=1017.432,10.106,-120.894,-24.190,21.513,-42.731
C05329=1017.431,10.483,-120.926,-24.191,21.513,-42.726
C05330=1017.430,10.864,-120.958,-24.191,21.513,-42.722
C05331=1017.429,11.248,-120.992,-24.192,21.512,-42.716
C05332=1017.428,11.633,-121.025,-24.192,21.511,-42.713
C05333=1017.427,12.019,-121.057,-24.193,21.512,-42.707
C05334=1017.426,12.406,-121.091,-24.193,21.510,-42.703
C05335=1017.425,12.792,-121.124,-24.194,21.510,-42.698
C05336=1017.424,13.179,-121.157,-24.195,21.511,-42.693
C05337=1017.422,13.566,-121.190,-24.196,21.509,-42.689
C05338=1017.421,13.953,-121.224,-24.196,21.509,-42.683
C05339=1017.420,14.341,-121.257,-24.197,21.509,-42.680
C05340=1017.419,14.729,-121.290,-24.198,21.508,-42.674
C05341=1017.418,15.118,-121.324,-24.198,21.508,-42.670
C05342=1017.416,15.507,-121.358,-24.199,21.507,-42.665
C05343=1017.415,15.898,-121.392,-24.200,21.507,-42.659
C05344=1017.414,16.289,-121.425,-24.200,21.506,-42.656
C05345=1017.412,16.680,-121.459,-24.201,21.506,-42.650
C05346=1017.411,17.072,-121.493,-24.201,21.505,-42.646
C05347=1017.410,17.466,-121.527,-24.202,21.505,-42.641
C05348=1017.409,17.860,-121.560,-24.203,21.505,-42.635
C05349=1017.408,18.255,-121.595,-24.203,21.504,-42.632
C05350=1017.406,18.652,-121.629,-24.204,21.503,-42.626
C05351=1017.405,19.048,-121.664,-24.205,21.503,-42.622
C05352=1017.403,19.445,-121.697,-24.205,21.503,-42.617
C05353=1017.402,19.656,-121.716,-24.206,21.503,-42.613
C05354=1017.401,19.893,-121.737,-24.206,21.502,-42.610
C05355=1017.401,20.158,-121.760,-24.207,21.503,-42.606
C05356=1017.400,20.445,-121.785,-24.207,21.501,-42.604
C05357=1017.399,20.742,-121.811,-24.207,21.501,-42.602
C05358=1017.398,21.033,-121.836,-24.208,21.502,-42.599
C05359=1017.396,21.306,-121.859,-24.208,21.501,-42.597
C05360=1017.396,21.550,-121.881,-24.209,21.501,-42.593
C05361=1017.395,21.964,-121.917,-24.210,21.501,-42.586
C05362=1017.393,22.339,-121.949,-24.210,21.500,-42.584
C05363=1017.392,22.660,-121.977,-24.211,21.500,-42.580
C05364=1017.390,22.927,-122.000,-24.211,21.500,-42.577
C05365=1017.389,23.158,-122.021,-24.211,21.499,-42.573
C05366=1017.389,23.393,-122.041,-24.212,21.498,-42.567
C05367=1017.388,23.665,-122.065,-24.213,21.498,-42.564
C05368=1017.386,23.995,-122.093,-24.213,21.498,-42.562
C05369=1017.385,24.378,-122.126,-24.213,21.497,-42.558
C05370=1017.383,24.777,-122.161,-24.214,21.497,-42.553
C05371=1017.382,25.176,-122.196,-24.215,21.497,-42.549
C05372=1017.380,25.575,-122.231,-24.215,21.496,-42.543
